Yaskawa INFORM job: A_ROOF_UPPER_0614_2_PAINT_64.JBI

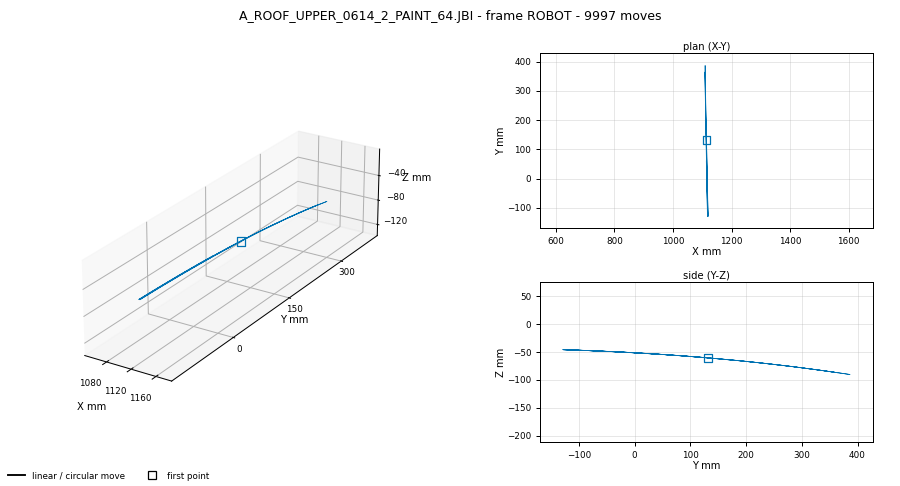
[picture p0: tool path of A_ROOF_UPPER_0614_2_PAINT_64.JBI in frame ROBOT, 9997 of 9997 moves have a stored position in this frame; points joined in program order, loops and branches not executed]
/JOB
//NAME A_ROOF_UPPER_0614_2_PAINT64
//POS
///NPOS 9997,0,0,0,0,0
///TOOL 1
///USER 0
///POSTYPE ROBOT
///RECTAN
///RCONF 1,0,0,0,0,0,0,0,0,0,0,0,0,0,0,0,0,0,0,0,0,0,0,0
C00000=1114.594,132.170,-60.301,-179.597,8.502,149.525
C00001=1114.597,131.955,-60.283,-179.599,8.499,149.525
C00002=1114.601,131.742,-60.265,-179.601,8.496,149.525
C00003=1114.606,131.528,-60.248,-179.602,8.493,149.525
C00004=1114.610,131.279,-60.226,-179.603,8.490,149.524
C00005=1114.614,131.030,-60.206,-179.605,8.487,149.524
C00006=1114.619,130.781,-60.185,-179.607,8.483,149.524
C00007=1114.624,130.532,-60.164,-179.609,8.480,149.523
C00008=1114.629,130.282,-60.143,-179.610,8.477,149.523
C00009=1114.634,130.034,-60.122,-179.613,8.473,149.523
C00010=1114.638,129.785,-60.101,-179.614,8.470,149.523
C00011=1114.643,129.535,-60.080,-179.616,8.467,149.522
C00012=1114.647,129.286,-60.059,-179.618,8.463,149.522
C00013=1114.653,129.037,-60.039,-179.619,8.460,149.522
C00014=1114.657,128.788,-60.018,-179.621,8.457,149.521
C00015=1114.662,128.539,-59.996,-179.623,8.453,149.521
C00016=1114.666,128.290,-59.976,-179.624,8.450,149.521
C00017=1114.671,128.041,-59.955,-179.626,8.447,149.521
C00018=1114.676,127.792,-59.935,-179.628,8.443,149.520
C00019=1114.681,127.543,-59.914,-179.630,8.440,149.520
C00020=1114.685,127.294,-59.893,-179.631,8.437,149.520
C00021=1114.691,127.044,-59.872,-179.634,8.433,149.519
C00022=1114.695,126.795,-59.852,-179.635,8.430,149.519
C00023=1114.700,126.547,-59.832,-179.637,8.427,149.519
C00024=1114.704,126.297,-59.810,-179.639,8.423,149.519
C00025=1114.709,126.048,-59.790,-179.640,8.420,149.518
C00026=1114.714,125.798,-59.769,-179.642,8.417,149.518
C00027=1114.718,125.549,-59.749,-179.644,8.413,149.518
C00028=1114.723,125.300,-59.728,-179.646,8.409,149.517
C00029=1114.728,125.051,-59.707,-179.647,8.407,149.517
C00030=1114.732,124.802,-59.687,-179.649,8.403,149.517
C00031=1114.737,124.553,-59.666,-179.651,8.400,149.517
C00032=1114.742,124.304,-59.646,-179.652,8.397,149.516
C00033=1114.746,124.055,-59.625,-179.655,8.393,149.516
C00034=1114.751,123.806,-59.604,-179.657,8.390,149.516
C00035=1114.756,123.557,-59.584,-179.658,8.387,149.516
C00036=1114.760,123.308,-59.564,-179.660,8.383,149.515
C00037=1114.765,123.059,-59.543,-179.662,8.380,149.515
C00038=1114.770,122.810,-59.522,-179.663,8.377,149.515
C00039=1114.774,122.561,-59.502,-179.665,8.373,149.515
C00040=1114.780,122.311,-59.482,-179.667,8.370,149.514
C00041=1114.784,122.062,-59.461,-179.669,8.366,149.514
C00042=1114.789,121.813,-59.441,-179.670,8.363,149.514
C00043=1114.794,121.564,-59.420,-179.672,8.360,149.513
C00044=1114.798,121.315,-59.399,-179.674,8.356,149.513
C00045=1114.803,121.066,-59.379,-179.675,8.353,149.513
C00046=1114.808,120.816,-59.359,-179.678,8.350,149.512
C00047=1114.813,120.567,-59.338,-179.680,8.346,149.512
C00048=1114.818,120.319,-59.318,-179.682,8.343,149.512
C00049=1114.822,120.070,-59.298,-179.683,8.340,149.512
C00050=1114.827,119.820,-59.278,-179.685,8.336,149.511
C00051=1114.832,119.571,-59.257,-179.687,8.333,149.511
C00052=1114.836,119.357,-59.240,-179.688,8.330,149.511
C00053=1114.839,119.143,-59.223,-179.690,8.327,149.511
C00054=1114.843,118.929,-59.205,-179.691,8.324,149.510
C00055=1114.848,118.715,-59.188,-179.693,8.321,149.510
C00056=1114.852,118.502,-59.171,-179.695,8.318,149.510
C00057=1114.856,118.288,-59.153,-179.696,8.315,149.510
C00058=1114.860,118.073,-59.135,-179.697,8.312,149.509
C00059=1114.864,117.860,-59.118,-179.698,8.310,149.509
C00060=1114.869,117.610,-59.098,-179.701,8.306,149.509
C00061=1114.873,117.361,-59.078,-179.703,8.303,149.509
C00062=1114.878,117.113,-59.058,-179.705,8.299,149.508
C00063=1114.883,116.863,-59.038,-179.706,8.296,149.508
C00064=1114.888,116.614,-59.017,-179.708,8.293,149.508
C00065=1114.893,116.364,-58.998,-179.710,8.289,149.508
C00066=1114.897,116.115,-58.977,-179.712,8.286,149.507
C00067=1114.902,115.867,-58.957,-179.713,8.282,149.507
C00068=1114.907,115.617,-58.937,-179.715,8.279,149.507
C00069=1114.912,115.369,-58.917,-179.717,8.275,149.506
C00070=1114.916,115.119,-58.898,-179.719,8.272,149.506
C00071=1114.921,114.870,-58.877,-179.721,8.268,149.506
C00072=1114.926,114.621,-58.858,-179.722,8.265,149.506
C00073=1114.930,114.372,-58.837,-179.724,8.262,149.505
C00074=1114.936,114.122,-58.817,-179.726,8.258,149.505
C00075=1114.941,113.874,-58.797,-179.728,8.254,149.505
C00076=1114.945,113.624,-58.777,-179.730,8.251,149.504
C00077=1114.950,113.375,-58.757,-179.731,8.248,149.504
C00078=1114.954,113.125,-58.737,-179.733,8.244,149.504
C00079=1114.959,112.876,-58.718,-179.735,8.241,149.504
C00080=1114.964,112.628,-58.698,-179.737,8.237,149.503
C00081=1114.969,112.378,-58.678,-179.739,8.233,149.503
C00082=1114.973,112.129,-58.658,-179.740,8.231,149.503
C00083=1114.978,111.880,-58.638,-179.742,8.227,149.502
C00084=1114.984,111.631,-58.619,-179.744,8.223,149.502
C00085=1114.988,111.382,-58.598,-179.746,8.220,149.502
C00086=1114.993,111.132,-58.579,-179.747,8.216,149.501
C00087=1114.997,110.883,-58.558,-179.749,8.213,149.501
C00088=1115.002,110.634,-58.539,-179.752,8.209,149.501
C00089=1115.007,110.385,-58.519,-179.754,8.206,149.501
C00090=1115.012,110.135,-58.500,-179.756,8.202,149.501
C00091=1115.016,109.886,-58.479,-179.758,8.199,149.500
C00092=1115.022,109.637,-58.460,-179.760,8.194,149.500
C00093=1115.026,109.388,-58.441,-179.762,8.190,149.500
C00094=1115.030,109.139,-58.421,-179.764,8.187,149.499
C00095=1115.036,108.890,-58.401,-179.766,8.183,149.499
C00096=1115.040,108.641,-58.382,-179.768,8.180,149.499
C00097=1115.045,108.391,-58.362,-179.770,8.176,149.499
C00098=1115.050,108.142,-58.343,-179.772,8.172,149.498
C00099=1115.055,107.893,-58.322,-179.775,8.168,149.498
C00100=1115.060,107.644,-58.303,-179.777,8.165,149.498
C00101=1115.064,107.395,-58.284,-179.778,8.161,149.497
C00102=1115.069,107.146,-58.264,-179.780,8.157,149.497
C00103=1115.074,106.896,-58.245,-179.782,8.154,149.497
C00104=1115.078,106.647,-58.225,-179.785,8.149,149.497
C00105=1115.083,106.398,-58.205,-179.787,8.146,149.496
C00106=1115.088,106.149,-58.185,-179.788,8.142,149.496
C00107=1115.093,105.900,-58.167,-179.790,8.138,149.496
C00108=1115.097,105.686,-58.150,-179.792,8.135,149.495
C00109=1115.101,105.472,-58.133,-179.793,8.132,149.495
C00110=1115.105,105.258,-58.116,-179.795,8.128,149.495
C00111=1115.110,105.043,-58.100,-179.797,8.125,149.495
C00112=1115.113,104.830,-58.083,-179.799,8.122,149.494
C00113=1115.118,104.616,-58.066,-179.800,8.119,149.494
C00114=1115.122,104.401,-58.050,-179.802,8.115,149.494
C00115=1115.126,104.188,-58.033,-179.803,8.113,149.493
C00116=1115.130,103.938,-58.014,-179.805,8.109,149.493
C00117=1115.135,103.689,-57.994,-179.807,8.105,149.493
C00118=1115.140,103.440,-57.975,-179.809,8.101,149.492
C00119=1115.144,103.191,-57.956,-179.811,8.097,149.492
C00120=1115.150,102.941,-57.937,-179.813,8.093,149.492
C00121=1115.155,102.692,-57.917,-179.814,8.089,149.491
C00122=1115.160,102.443,-57.898,-179.817,8.086,149.491
C00123=1115.164,102.194,-57.879,-179.818,8.082,149.491
C00124=1115.169,101.944,-57.859,-179.820,8.078,149.490
C00125=1115.174,101.695,-57.840,-179.822,8.074,149.490
C00126=1115.178,101.446,-57.821,-179.823,8.071,149.490
C00127=1115.183,101.197,-57.802,-179.825,8.067,149.489
C00128=1115.188,100.947,-57.782,-179.827,8.063,149.489
C00129=1115.193,100.699,-57.763,-179.829,8.059,149.488
C00130=1115.198,100.449,-57.744,-179.830,8.055,149.488
C00131=1115.202,100.200,-57.726,-179.832,8.052,149.488
C00132=1115.207,99.951,-57.706,-179.833,8.048,149.487
C00133=1115.212,99.702,-57.687,-179.836,8.044,149.487
C00134=1115.216,99.452,-57.668,-179.837,8.040,149.486
C00135=1115.222,99.203,-57.649,-179.839,8.036,149.486
C00136=1115.226,98.954,-57.630,-179.840,8.032,149.486
C00137=1115.231,98.705,-57.611,-179.842,8.029,149.485
C00138=1115.235,98.456,-57.592,-179.844,8.025,149.485
C00139=1115.241,98.206,-57.573,-179.846,8.021,149.485
C00140=1115.246,97.957,-57.554,-179.847,8.017,149.484
C00141=1115.250,97.708,-57.535,-179.849,8.013,149.484
C00142=1115.256,97.458,-57.516,-179.850,8.010,149.483
C00143=1115.260,97.209,-57.497,-179.852,8.006,149.483
C00144=1115.265,96.960,-57.478,-179.854,8.002,149.482
C00145=1115.270,96.710,-57.460,-179.855,7.998,149.482
C00146=1115.275,96.462,-57.440,-179.857,7.994,149.481
C00147=1115.279,96.212,-57.421,-179.858,7.990,149.481
C00148=1115.285,95.963,-57.403,-179.860,7.986,149.481
C00149=1115.289,95.714,-57.384,-179.862,7.982,149.480
C00150=1115.293,95.465,-57.365,-179.863,7.978,149.480
C00151=1115.298,95.215,-57.346,-179.865,7.975,149.479
C00152=1115.303,94.966,-57.327,-179.866,7.971,149.479
C00153=1115.309,94.717,-57.309,-179.868,7.967,149.478
C00154=1115.313,94.468,-57.290,-179.870,7.963,149.478
C00155=1115.318,94.218,-57.271,-179.871,7.959,149.478
C00156=1115.322,93.969,-57.252,-179.872,7.956,149.477
C00157=1115.328,93.719,-57.233,-179.874,7.952,149.477
C00158=1115.333,93.471,-57.215,-179.875,7.948,149.476
C00159=1115.337,93.221,-57.196,-179.877,7.944,149.476
C00160=1115.342,92.972,-57.177,-179.879,7.940,149.475
C00161=1115.347,92.723,-57.159,-179.880,7.936,149.475
C00162=1115.352,92.473,-57.139,-179.881,7.932,149.474
C00163=1115.357,92.224,-57.121,-179.883,7.928,149.474
C00164=1115.361,92.010,-57.105,-179.884,7.925,149.473
C00165=1115.364,91.796,-57.089,-179.885,7.922,149.473
C00166=1115.368,91.582,-57.073,-179.886,7.919,149.473
C00167=1115.373,91.368,-57.057,-179.888,7.915,149.472
C00168=1115.378,91.153,-57.041,-179.889,7.912,149.472
C00169=1115.381,90.939,-57.025,-179.890,7.909,149.472
C00170=1115.385,90.725,-57.009,-179.891,7.905,149.471
C00171=1115.390,90.512,-56.994,-179.892,7.902,149.471
C00172=1115.395,90.262,-56.975,-179.894,7.898,149.470
C00173=1115.400,90.012,-56.957,-179.896,7.894,149.470
C00174=1115.404,89.764,-56.938,-179.897,7.891,149.469
C00175=1115.409,89.514,-56.920,-179.898,7.887,149.469
C00176=1115.414,89.265,-56.901,-179.899,7.883,149.468
C00177=1115.419,89.016,-56.882,-179.901,7.879,149.468
C00178=1115.423,88.766,-56.864,-179.902,7.876,149.467
C00179=1115.429,88.517,-56.845,-179.903,7.872,149.467
C00180=1115.433,88.268,-56.827,-179.905,7.868,149.466
C00181=1115.438,88.019,-56.809,-179.906,7.864,149.466
C00182=1115.443,87.769,-56.790,-179.907,7.861,149.465
C00183=1115.448,87.520,-56.771,-179.908,7.857,149.465
C00184=1115.453,87.271,-56.753,-179.910,7.853,149.464
C00185=1115.458,87.022,-56.735,-179.911,7.848,149.464
C00186=1115.462,86.772,-56.717,-179.912,7.845,149.463
C00187=1115.467,86.523,-56.699,-179.914,7.841,149.463
C00188=1115.472,86.274,-56.680,-179.915,7.837,149.462
C00189=1115.477,86.025,-56.662,-179.916,7.833,149.462
C00190=1115.482,85.775,-56.643,-179.917,7.830,149.461
C00191=1115.486,85.526,-56.625,-179.918,7.826,149.461
C00192=1115.491,85.276,-56.607,-179.920,7.822,149.460
C00193=1115.496,85.028,-56.589,-179.920,7.819,149.460
C00194=1115.501,84.778,-56.570,-179.922,7.815,149.459
C00195=1115.506,84.529,-56.552,-179.924,7.811,149.459
C00196=1115.511,84.279,-56.534,-179.924,7.807,149.458
C00197=1115.516,84.030,-56.516,-179.926,7.803,149.458
C00198=1115.521,83.781,-56.498,-179.927,7.799,149.457
C00199=1115.525,83.531,-56.479,-179.928,7.796,149.457
C00200=1115.530,83.282,-56.461,-179.929,7.792,149.456
C00201=1115.535,83.033,-56.443,-179.930,7.789,149.456
C00202=1115.540,82.784,-56.424,-179.932,7.785,149.455
C00203=1115.545,82.535,-56.406,-179.933,7.780,149.455
C00204=1115.549,82.285,-56.388,-179.934,7.777,149.454
C00205=1115.554,82.036,-56.370,-179.935,7.773,149.453
C00206=1115.559,81.786,-56.352,-179.936,7.770,149.453
C00207=1115.564,81.537,-56.334,-179.937,7.766,149.452
C00208=1115.569,81.288,-56.316,-179.938,7.762,149.452
C00209=1115.574,81.039,-56.298,-179.939,7.758,149.451
C00210=1115.578,80.789,-56.280,-179.941,7.754,149.451
C00211=1115.583,80.540,-56.262,-179.941,7.751,149.450
C00212=1115.588,80.291,-56.244,-179.943,7.747,149.450
C00213=1115.593,80.042,-56.226,-179.943,7.743,149.449
C00214=1115.598,79.792,-56.208,-179.945,7.740,149.449
C00215=1115.603,79.543,-56.190,-179.945,7.736,149.448
C00216=1115.608,79.293,-56.172,-179.946,7.732,149.447
C00217=1115.613,79.044,-56.154,-179.947,7.729,149.447
C00218=1115.617,78.794,-56.136,-179.948,7.724,149.446
C00219=1115.622,78.545,-56.118,-179.949,7.721,149.446
C00220=1115.627,78.332,-56.102,-179.950,7.718,149.445
C00221=1115.631,78.117,-56.087,-179.951,7.715,149.445
C00222=1115.635,77.902,-56.072,-179.952,7.712,149.444
C00223=1115.640,77.688,-56.057,-179.953,7.708,149.444
C00224=1115.643,77.474,-56.040,-179.954,7.705,149.444
C00225=1115.648,77.260,-56.025,-179.955,7.702,149.443
C00226=1115.651,77.046,-56.011,-179.955,7.699,149.442
C00227=1115.656,76.832,-55.995,-179.956,7.696,149.442
C00228=1115.661,76.582,-55.977,-179.958,7.692,149.442
C00229=1115.665,76.333,-55.959,-179.959,7.688,149.441
C00230=1115.670,76.084,-55.941,-179.960,7.683,149.440
C00231=1115.675,75.834,-55.923,-179.962,7.680,149.440
C00232=1115.680,75.585,-55.905,-179.964,7.676,149.440
C00233=1115.685,75.335,-55.888,-179.965,7.672,149.439
C00234=1115.690,75.086,-55.870,-179.966,7.667,149.439
C00235=1115.695,74.837,-55.852,-179.968,7.664,149.438
C00236=1115.699,74.588,-55.835,-179.969,7.660,149.438
C00237=1115.705,74.338,-55.817,-179.970,7.656,149.437
C00238=1115.710,74.089,-55.799,-179.971,7.652,149.437
C00239=1115.714,73.840,-55.781,-179.973,7.648,149.436
C00240=1115.719,73.591,-55.764,-179.975,7.644,149.436
C00241=1115.725,73.341,-55.746,-179.976,7.640,149.435
C00242=1115.729,73.092,-55.728,-179.977,7.636,149.435
C00243=1115.734,72.843,-55.711,-179.979,7.632,149.434
C00244=1115.739,72.593,-55.694,-179.980,7.628,149.434
C00245=1115.744,72.344,-55.676,-179.982,7.624,149.433
C00246=1115.749,72.095,-55.658,-179.983,7.620,149.433
C00247=1115.754,71.845,-55.640,-179.985,7.616,149.432
C00248=1115.758,71.596,-55.623,-179.986,7.612,149.432
C00249=1115.763,71.346,-55.606,-179.987,7.608,149.431
C00250=1115.768,71.097,-55.588,-179.988,7.605,149.431
C00251=1115.773,70.848,-55.570,-179.990,7.601,149.430
C00252=1115.778,70.599,-55.553,-179.991,7.597,149.430
C00253=1115.782,70.349,-55.535,-179.993,7.593,149.429
C00254=1115.788,70.100,-55.518,-179.994,7.589,149.429
C00255=1115.793,69.850,-55.500,-179.995,7.585,149.428
C00256=1115.797,69.601,-55.483,-179.997,7.581,149.428
C00257=1115.802,69.352,-55.465,-179.998,7.577,149.427
C00258=1115.807,69.102,-55.448,-180.000,7.573,149.427
C00259=1115.812,68.853,-55.430,179.999,7.569,149.426
C00260=1115.817,68.604,-55.414,179.997,7.565,149.426
C00261=1115.822,68.355,-55.396,179.997,7.561,149.425
C00262=1115.827,68.105,-55.378,179.995,7.558,149.425
C00263=1115.832,67.856,-55.361,179.994,7.554,149.424
C00264=1115.837,67.606,-55.344,179.993,7.549,149.424
C00265=1115.842,67.357,-55.326,179.991,7.545,149.423
C00266=1115.846,67.108,-55.309,179.989,7.542,149.423
C00267=1115.851,66.858,-55.292,179.988,7.537,149.422
C00268=1115.856,66.609,-55.274,179.987,7.533,149.422
C00269=1115.861,66.359,-55.257,179.985,7.529,149.421
C00270=1115.866,66.111,-55.240,179.984,7.525,149.421
C00271=1115.871,65.861,-55.223,179.983,7.522,149.420
C00272=1115.876,65.612,-55.206,179.982,7.518,149.420
C00273=1115.881,65.362,-55.188,179.980,7.514,149.419
C00274=1115.885,65.113,-55.171,179.979,7.510,149.419
C00275=1115.891,64.863,-55.154,179.978,7.506,149.418
C00276=1115.895,64.649,-55.139,179.977,7.502,149.418
C00277=1115.899,64.435,-55.124,179.975,7.499,149.417
C00278=1115.903,64.221,-55.110,179.974,7.495,149.417
C00279=1115.908,64.006,-55.095,179.973,7.492,149.416
C00280=1115.911,63.792,-55.080,179.972,7.488,149.416
C00281=1115.916,63.578,-55.065,179.971,7.485,149.415
C00282=1115.920,63.363,-55.050,179.970,7.482,149.415
C00283=1115.924,63.149,-55.036,179.968,7.478,149.415
C00284=1115.929,62.900,-55.018,179.967,7.474,149.414
C00285=1115.934,62.650,-55.002,179.966,7.470,149.413
C00286=1115.939,62.400,-54.984,179.965,7.467,149.413
C00287=1115.944,62.152,-54.968,179.964,7.463,149.412
C00288=1115.949,61.902,-54.950,179.962,7.459,149.412
C00289=1115.953,61.653,-54.933,179.960,7.455,149.412
C00290=1115.959,61.403,-54.916,179.959,7.451,149.411
C00291=1115.964,61.154,-54.900,179.958,7.447,149.410
C00292=1115.969,60.905,-54.883,179.957,7.442,149.410
C00293=1115.973,60.655,-54.866,179.955,7.438,149.409
C00294=1115.978,60.406,-54.849,179.954,7.434,149.409
C00295=1115.983,60.156,-54.831,179.953,7.431,149.408
C00296=1115.988,59.908,-54.815,179.952,7.427,149.408
C00297=1115.993,59.658,-54.798,179.950,7.423,149.407
C00298=1115.998,59.408,-54.781,179.949,7.419,149.407
C00299=1116.003,59.159,-54.764,179.948,7.415,149.406
C00300=1116.008,58.910,-54.748,179.946,7.411,149.406
C00301=1116.012,58.660,-54.731,179.945,7.406,149.405
C00302=1116.017,58.410,-54.714,179.944,7.403,149.405
C00303=1116.023,58.162,-54.697,179.943,7.399,149.404
C00304=1116.028,57.912,-54.680,179.942,7.395,149.404
C00305=1116.032,57.662,-54.663,179.940,7.391,149.403
C00306=1116.037,57.413,-54.647,179.939,7.387,149.402
C00307=1116.043,57.164,-54.630,179.938,7.383,149.402
C00308=1116.047,56.914,-54.613,179.936,7.379,149.401
C00309=1116.052,56.665,-54.596,179.935,7.374,149.401
C00310=1116.057,56.416,-54.580,179.934,7.370,149.400
C00311=1116.062,56.166,-54.563,179.933,7.367,149.400
C00312=1116.066,55.917,-54.546,179.932,7.363,149.399
C00313=1116.072,55.668,-54.529,179.930,7.359,149.399
C00314=1116.077,55.418,-54.513,179.929,7.355,149.398
C00315=1116.081,55.169,-54.496,179.928,7.351,149.398
C00316=1116.087,54.920,-54.479,179.926,7.347,149.397
C00317=1116.091,54.670,-54.462,179.925,7.342,149.396
C00318=1116.096,54.421,-54.446,179.924,7.338,149.396
C00319=1116.102,54.171,-54.430,179.923,7.335,149.395
C00320=1116.106,53.922,-54.413,179.922,7.331,149.395
C00321=1116.112,53.673,-54.397,179.920,7.327,149.394
C00322=1116.116,53.423,-54.380,179.919,7.323,149.394
C00323=1116.121,53.173,-54.363,179.918,7.319,149.393
C00324=1116.126,52.925,-54.346,179.916,7.315,149.393
C00325=1116.131,52.675,-54.330,179.915,7.310,149.392
C00326=1116.136,52.426,-54.314,179.915,7.307,149.391
C00327=1116.141,52.176,-54.297,179.913,7.303,149.391
C00328=1116.146,51.926,-54.280,179.912,7.299,149.390
C00329=1116.151,51.677,-54.265,179.910,7.295,149.390
C00330=1116.156,51.428,-54.248,179.909,7.290,149.389
C00331=1116.161,51.179,-54.232,179.908,7.286,149.389
C00332=1116.165,50.963,-54.217,179.907,7.283,149.388
C00333=1116.169,50.750,-54.203,179.906,7.280,149.388
C00334=1116.174,50.535,-54.189,179.905,7.276,149.387
C00335=1116.178,50.321,-54.175,179.904,7.273,149.387
C00336=1116.182,50.106,-54.160,179.903,7.269,149.386
C00337=1116.186,49.892,-54.146,179.902,7.265,149.386
C00338=1116.191,49.678,-54.132,179.901,7.262,149.385
C00339=1116.195,49.463,-54.119,179.900,7.259,149.385
C00340=1116.199,49.214,-54.102,179.899,7.255,149.384
C00341=1116.205,48.965,-54.086,179.898,7.250,149.384
C00342=1116.209,48.715,-54.070,179.896,7.247,149.383
C00343=1116.215,48.466,-54.053,179.895,7.242,149.383
C00344=1116.223,48.072,-54.028,179.893,7.236,149.382
C00345=1116.230,47.678,-54.002,179.892,7.230,149.381
C00346=1116.238,47.284,-53.976,179.890,7.224,149.380
C00347=1116.245,46.890,-53.950,179.888,7.217,149.379
C00348=1116.251,46.641,-53.935,179.887,7.213,149.378
C00349=1116.255,46.391,-53.918,179.886,7.209,149.378
C00350=1116.260,46.142,-53.902,179.885,7.204,149.377
C00351=1116.266,45.893,-53.886,179.883,7.200,149.377
C00352=1116.270,45.643,-53.870,179.882,7.196,149.376
C00353=1116.276,45.394,-53.854,179.881,7.193,149.375
C00354=1116.280,45.145,-53.837,179.880,7.188,149.375
C00355=1116.286,44.895,-53.822,179.879,7.184,149.374
C00356=1116.290,44.646,-53.805,179.878,7.180,149.374
C00357=1116.295,44.396,-53.789,179.877,7.176,149.373
C00358=1116.300,44.146,-53.773,179.875,7.172,149.373
C00359=1116.305,43.897,-53.757,179.874,7.168,149.372
C00360=1116.310,43.647,-53.741,179.874,7.164,149.371
C00361=1116.315,43.399,-53.725,179.873,7.160,149.371
C00362=1116.320,43.148,-53.709,179.871,7.156,149.370
C00363=1116.325,42.900,-53.693,179.870,7.152,149.370
C00364=1116.330,42.650,-53.677,179.869,7.147,149.369
C00365=1116.335,42.400,-53.661,179.868,7.143,149.368
C00366=1116.340,42.151,-53.645,179.867,7.139,149.368
C00367=1116.345,41.901,-53.629,179.866,7.135,149.367
C00368=1116.350,41.652,-53.613,179.865,7.131,149.367
C00369=1116.356,41.403,-53.597,179.864,7.127,149.366
C00370=1116.360,41.153,-53.581,179.863,7.123,149.365
C00371=1116.366,40.904,-53.565,179.861,7.118,149.365
C00372=1116.369,40.654,-53.549,179.860,7.114,149.364
C00373=1116.375,40.405,-53.534,179.859,7.110,149.364
C00374=1116.380,40.156,-53.518,179.858,7.106,149.363
C00375=1116.385,39.906,-53.502,179.857,7.102,149.362
C00376=1116.390,39.657,-53.486,179.856,7.098,149.362
C00377=1116.395,39.407,-53.470,179.855,7.094,149.361
C00378=1116.400,39.157,-53.454,179.854,7.090,149.360
C00379=1116.405,38.909,-53.439,179.853,7.085,149.360
C00380=1116.410,38.659,-53.423,179.852,7.081,149.359
C00381=1116.415,38.409,-53.407,179.850,7.077,149.359
C00382=1116.420,38.160,-53.392,179.850,7.073,149.358
C00383=1116.426,37.910,-53.376,179.849,7.069,149.357
C00384=1116.430,37.661,-53.359,179.848,7.065,149.357
C00385=1116.435,37.412,-53.344,179.847,7.060,149.356
C00386=1116.440,37.162,-53.329,179.845,7.056,149.356
C00387=1116.445,36.912,-53.313,179.844,7.052,149.355
C00388=1116.451,36.628,-53.295,179.844,7.047,149.354
C00389=1116.456,36.344,-53.277,179.842,7.042,149.353
C00390=1116.462,36.059,-53.259,179.841,7.038,149.353
C00391=1116.468,35.775,-53.241,179.840,7.033,149.352
C00392=1116.472,35.525,-53.226,179.839,7.029,149.351
C00393=1116.478,35.275,-53.210,179.838,7.025,149.351
C00394=1116.483,35.026,-53.195,179.837,7.020,149.350
C00395=1116.488,34.777,-53.179,179.836,7.016,149.349
C00396=1116.492,34.527,-53.164,179.834,7.012,149.349
C00397=1116.498,34.277,-53.148,179.833,7.008,149.348
C00398=1116.503,34.029,-53.132,179.832,7.004,149.347
C00399=1116.508,33.778,-53.116,179.831,6.999,149.347
C00400=1116.512,33.529,-53.101,179.831,6.996,149.346
C00401=1116.518,33.280,-53.085,179.830,6.991,149.346
C00402=1116.523,33.031,-53.070,179.829,6.987,149.345
C00403=1116.528,32.781,-53.055,179.828,6.983,149.344
C00404=1116.533,32.531,-53.039,179.827,6.978,149.344
C00405=1116.538,32.282,-53.023,179.825,6.974,149.343
C00406=1116.543,32.032,-53.009,179.825,6.969,149.342
C00407=1116.548,31.783,-52.993,179.824,6.965,149.341
C00408=1116.552,31.533,-52.978,179.823,6.962,149.341
C00409=1116.558,31.284,-52.962,179.822,6.957,149.340
C00410=1116.563,31.034,-52.947,179.821,6.953,149.339
C00411=1116.568,30.785,-52.932,179.820,6.949,149.339
C00412=1116.573,30.536,-52.916,179.819,6.944,149.338
C00413=1116.578,30.286,-52.900,179.818,6.940,149.337
C00414=1116.583,30.037,-52.885,179.817,6.936,149.337
C00415=1116.588,29.787,-52.870,179.816,6.931,149.336
C00416=1116.593,29.538,-52.855,179.816,6.928,149.335
C00417=1116.598,29.288,-52.840,179.814,6.924,149.335
C00418=1116.602,29.038,-52.825,179.814,6.919,149.334
C00419=1116.608,28.789,-52.809,179.813,6.915,149.333
C00420=1116.613,28.539,-52.793,179.812,6.910,149.333
C00421=1116.618,28.290,-52.778,179.811,6.906,149.332
C00422=1116.623,28.040,-52.764,179.810,6.902,149.331
C00423=1116.628,27.791,-52.749,179.809,6.897,149.331
C00424=1116.634,27.542,-52.733,179.808,6.893,149.330
C00425=1116.638,27.292,-52.718,179.807,6.888,149.329
C00426=1116.643,27.043,-52.702,179.807,6.885,149.329
C00427=1116.648,26.793,-52.688,179.805,6.880,149.328
C00428=1116.653,26.544,-52.672,179.804,6.876,149.327
C00429=1116.658,26.294,-52.657,179.803,6.872,149.327
C00430=1116.663,26.045,-52.642,179.803,6.867,149.326
C00431=1116.668,25.795,-52.627,179.802,6.863,149.325
C00432=1116.674,25.546,-52.612,179.801,6.859,149.324
C00433=1116.678,25.297,-52.597,179.800,6.854,149.324
C00434=1116.683,25.046,-52.581,179.799,6.850,149.323
C00435=1116.688,24.797,-52.566,179.799,6.846,149.322
C00436=1116.693,24.548,-52.551,179.798,6.842,149.322
C00437=1116.698,24.298,-52.537,179.797,6.837,149.321
C00438=1116.703,24.049,-52.522,179.796,6.833,149.320
C00439=1116.708,23.799,-52.506,179.795,6.828,149.319
C00440=1116.712,23.585,-52.494,179.794,6.825,149.319
C00441=1116.717,23.370,-52.481,179.793,6.821,149.318
C00442=1116.721,23.155,-52.468,179.793,6.817,149.318
C00443=1116.726,22.942,-52.455,179.791,6.813,149.317
C00444=1116.730,22.727,-52.442,179.791,6.810,149.316
C00445=1116.734,22.512,-52.429,179.791,6.806,149.316
C00446=1116.739,22.297,-52.417,179.790,6.802,149.315
C00447=1116.743,22.082,-52.404,179.789,6.798,149.314
C00448=1116.748,21.833,-52.389,179.788,6.794,149.314
C00449=1116.753,21.583,-52.374,179.787,6.789,149.313
C00450=1116.758,21.334,-52.359,179.786,6.785,149.312
C00451=1116.763,21.085,-52.344,179.785,6.780,149.311
C00452=1116.768,20.835,-52.329,179.784,6.776,149.311
C00453=1116.773,20.586,-52.314,179.784,6.771,149.310
C00454=1116.778,20.336,-52.300,179.783,6.768,149.309
C00455=1116.783,20.087,-52.285,179.783,6.763,149.308
C00456=1116.788,19.837,-52.270,179.782,6.759,149.308
C00457=1116.794,19.587,-52.255,179.781,6.755,149.307
C00458=1116.798,19.338,-52.240,179.780,6.750,149.306
C00459=1116.803,19.088,-52.226,179.779,6.746,149.306
C00460=1116.809,18.839,-52.211,179.779,6.741,149.305
C00461=1116.814,18.589,-52.196,179.778,6.737,149.304
C00462=1116.818,18.340,-52.181,179.777,6.732,149.303
C00463=1116.823,18.090,-52.167,179.776,6.728,149.303
C00464=1116.829,17.840,-52.152,179.775,6.723,149.302
C00465=1116.833,17.591,-52.137,179.774,6.718,149.301
C00466=1116.838,17.342,-52.123,179.773,6.714,149.300
C00467=1116.843,17.093,-52.108,179.773,6.709,149.299
C00468=1116.849,16.842,-52.093,179.772,6.706,149.299
C00469=1116.854,16.593,-52.079,179.772,6.701,149.298
C00470=1116.859,16.344,-52.064,179.771,6.697,149.297
C00471=1116.864,16.095,-52.050,179.770,6.692,149.296
C00472=1116.869,15.845,-52.036,179.770,6.687,149.295
C00473=1116.874,15.596,-52.020,179.769,6.683,149.295
C00474=1116.879,15.346,-52.006,179.768,6.678,149.294
C00475=1116.884,15.096,-51.991,179.767,6.674,149.293
C00476=1116.889,14.846,-51.977,179.766,6.669,149.292
C00477=1116.894,14.597,-51.962,179.765,6.665,149.292
C00478=1116.899,14.348,-51.948,179.765,6.660,149.291
C00479=1116.904,14.098,-51.933,179.764,6.656,149.290
C00480=1116.910,13.849,-51.919,179.763,6.651,149.289
C00481=1116.915,13.600,-51.904,179.763,6.647,149.288
C00482=1116.920,13.350,-51.890,179.762,6.642,149.288
C00483=1116.925,13.100,-51.875,179.761,6.638,149.287
C00484=1116.929,12.850,-51.861,179.761,6.633,149.286
C00485=1116.934,12.601,-51.846,179.760,6.629,149.285
C00486=1116.940,12.351,-51.831,179.759,6.624,149.285
C00487=1116.945,12.102,-51.817,179.758,6.619,149.284
C00488=1116.950,11.853,-51.803,179.757,6.615,149.283
C00489=1116.955,11.603,-51.789,179.757,6.610,149.282
C00490=1116.960,11.353,-51.775,179.757,6.606,149.281
C00491=1116.965,11.103,-51.760,179.756,6.601,149.280
C00492=1116.970,10.854,-51.745,179.755,6.597,149.280
C00493=1116.975,10.605,-51.731,179.755,6.592,149.279
C00494=1116.980,10.356,-51.717,179.754,6.588,149.278
C00495=1116.985,10.106,-51.703,179.753,6.583,149.277
C00496=1116.989,9.891,-51.690,179.753,6.579,149.276
C00497=1116.994,9.676,-51.678,179.752,6.575,149.276
C00498=1116.999,9.462,-51.666,179.751,6.571,149.275
C00499=1117.002,9.247,-51.654,179.751,6.567,149.274
C00500=1117.007,9.032,-51.641,179.751,6.563,149.274
C00501=1117.012,8.818,-51.629,179.750,6.559,149.273
C00502=1117.016,8.603,-51.617,179.749,6.556,149.272
C00503=1117.020,8.388,-51.604,179.749,6.551,149.271
C00504=1117.026,8.139,-51.590,179.748,6.547,149.271
C00505=1117.030,7.890,-51.576,179.747,6.542,149.270
C00506=1117.035,7.640,-51.562,179.747,6.538,149.269
C00507=1117.040,7.390,-51.548,179.747,6.533,149.268
C00508=1117.045,7.141,-51.534,179.746,6.528,149.267
C00509=1117.050,6.891,-51.520,179.746,6.524,149.266
C00510=1117.055,6.642,-51.505,179.745,6.519,149.265
C00511=1117.060,6.392,-51.491,179.744,6.515,149.265
C00512=1117.065,6.142,-51.477,179.744,6.510,149.264
C00513=1117.071,5.893,-51.464,179.743,6.505,149.263
C00514=1117.076,5.643,-51.449,179.743,6.501,149.262
C00515=1117.081,5.393,-51.435,179.743,6.497,149.261
C00516=1117.087,5.144,-51.421,179.742,6.492,149.260
C00517=1117.092,4.895,-51.407,179.741,6.488,149.260
C00518=1117.097,4.645,-51.393,179.741,6.483,149.259
C00519=1117.102,4.395,-51.378,179.740,6.478,149.258
C00520=1117.106,4.146,-51.365,179.739,6.473,149.257
C00521=1117.111,3.897,-51.351,179.739,6.469,149.256
C00522=1117.117,3.646,-51.337,179.739,6.465,149.255
C00523=1117.122,3.397,-51.323,179.738,6.460,149.255
C00524=1117.127,3.148,-51.309,179.737,6.456,149.254
C00525=1117.132,2.898,-51.295,179.737,6.451,149.253
C00526=1117.137,2.648,-51.281,179.736,6.446,149.252
C00527=1117.142,2.400,-51.267,179.735,6.442,149.251
C00528=1117.147,2.149,-51.254,179.735,6.437,149.250
C00529=1117.152,1.900,-51.239,179.734,6.433,149.249
C00530=1117.158,1.651,-51.225,179.734,6.429,149.249
C00531=1117.162,1.401,-51.211,179.733,6.424,149.248
C00532=1117.167,1.151,-51.198,179.733,6.420,149.247
C00533=1117.173,0.902,-51.184,179.732,6.415,149.246
C00534=1117.178,0.652,-51.170,179.732,6.410,149.245
C00535=1117.182,0.402,-51.156,179.731,6.406,149.245
C00536=1117.188,0.153,-51.143,179.730,6.401,149.244
C00537=1117.193,-0.097,-51.129,179.730,6.396,149.243
C00538=1117.198,-0.346,-51.115,179.730,6.392,149.242
C00539=1117.203,-0.596,-51.101,179.729,6.388,149.241
C00540=1117.208,-0.846,-51.087,179.728,6.383,149.240
C00541=1117.213,-1.094,-51.074,179.728,6.379,149.239
C00542=1117.218,-1.345,-51.060,179.727,6.374,149.239
C00543=1117.223,-1.594,-51.046,179.726,6.370,149.238
C00544=1117.229,-1.843,-51.032,179.726,6.365,149.237
C00545=1117.233,-2.093,-51.019,179.725,6.360,149.236
C00546=1117.239,-2.342,-51.005,179.725,6.357,149.235
C00547=1117.244,-2.592,-50.991,179.724,6.352,149.235
C00548=1117.248,-2.842,-50.978,179.724,6.347,149.234
C00549=1117.254,-3.091,-50.964,179.723,6.343,149.233
C00550=1117.259,-3.342,-50.950,179.722,6.338,149.232
C00551=1117.265,-3.591,-50.937,179.722,6.333,149.231
C00552=1117.269,-3.806,-50.925,179.721,6.330,149.231
C00553=1117.273,-4.020,-50.913,179.720,6.326,149.230
C00554=1117.278,-4.235,-50.901,179.720,6.322,149.229
C00555=1117.282,-4.450,-50.890,179.720,6.318,149.228
C00556=1117.287,-4.665,-50.878,179.719,6.314,149.228
C00557=1117.291,-4.879,-50.866,179.719,6.310,149.227
C00558=1117.295,-5.094,-50.854,179.718,6.307,149.226
C00559=1117.300,-5.309,-50.843,179.717,6.302,149.226
C00560=1117.305,-5.559,-50.830,179.717,6.298,149.225
C00561=1117.310,-5.808,-50.816,179.716,6.293,149.224
C00562=1117.315,-6.058,-50.803,179.716,6.289,149.223
C00563=1117.320,-6.307,-50.789,179.715,6.285,149.222
C00564=1117.325,-6.557,-50.776,179.715,6.280,149.221
C00565=1117.330,-6.806,-50.762,179.714,6.276,149.221
C00566=1117.336,-7.056,-50.749,179.713,6.271,149.220
C00567=1117.340,-7.305,-50.735,179.713,6.266,149.219
C00568=1117.346,-7.555,-50.722,179.712,6.261,149.218
C00569=1117.351,-7.805,-50.708,179.711,6.257,149.218
C00570=1117.356,-8.054,-50.695,179.711,6.252,149.217
C00571=1117.361,-8.304,-50.682,179.710,6.248,149.216
C00572=1117.366,-8.553,-50.668,179.709,6.243,149.215
C00573=1117.372,-8.803,-50.655,179.709,6.239,149.214
C00574=1117.376,-9.052,-50.641,179.709,6.235,149.213
C00575=1117.382,-9.302,-50.628,179.708,6.230,149.213
C00576=1117.386,-9.552,-50.615,179.707,6.226,149.212
C00577=1117.392,-9.801,-50.601,179.707,6.221,149.211
C00578=1117.396,-10.051,-50.588,179.706,6.216,149.210
C00579=1117.402,-10.300,-50.575,179.705,6.212,149.209
C00580=1117.406,-10.550,-50.561,179.705,6.207,149.208
C00581=1117.412,-10.799,-50.548,179.704,6.202,149.207
C00582=1117.417,-11.049,-50.535,179.703,6.198,149.207
C00583=1117.423,-11.299,-50.522,179.703,6.193,149.206
C00584=1117.427,-11.549,-50.508,179.702,6.189,149.205
C00585=1117.433,-11.798,-50.495,179.702,6.184,149.204
C00586=1117.438,-12.047,-50.483,179.701,6.179,149.203
C00587=1117.443,-12.298,-50.469,179.700,6.175,149.203
C00588=1117.448,-12.546,-50.456,179.700,6.170,149.202
C00589=1117.452,-12.796,-50.443,179.699,6.166,149.201
C00590=1117.458,-13.046,-50.430,179.698,6.161,149.200
C00591=1117.463,-13.295,-50.417,179.698,6.156,149.199
C00592=1117.468,-13.545,-50.403,179.697,6.151,149.198
C00593=1117.473,-13.794,-50.390,179.696,6.147,149.198
C00594=1117.478,-14.044,-50.377,179.696,6.142,149.197
C00595=1117.484,-14.294,-50.364,179.695,6.138,149.196
C00596=1117.489,-14.543,-50.351,179.695,6.133,149.195
C00597=1117.494,-14.794,-50.338,179.694,6.129,149.194
C00598=1117.499,-15.042,-50.324,179.693,6.124,149.193
C00599=1117.504,-15.292,-50.312,179.693,6.119,149.193
C00600=1117.509,-15.542,-50.298,179.692,6.114,149.192
C00601=1117.515,-15.791,-50.286,179.691,6.110,149.191
C00602=1117.519,-16.041,-50.273,179.691,6.105,149.190
C00603=1117.525,-16.291,-50.260,179.690,6.101,149.189
C00604=1117.530,-16.540,-50.247,179.690,6.096,149.188
C00605=1117.535,-16.790,-50.234,179.689,6.092,149.188
C00606=1117.540,-17.040,-50.221,179.689,6.087,149.187
C00607=1117.546,-17.289,-50.208,179.688,6.082,149.186
C00608=1117.550,-17.505,-50.197,179.688,6.079,149.185
C00609=1117.554,-17.719,-50.186,179.687,6.074,149.184
C00610=1117.559,-17.933,-50.174,179.687,6.070,149.184
C00611=1117.563,-18.149,-50.163,179.686,6.066,149.183
C00612=1117.568,-18.364,-50.152,179.685,6.062,149.182
C00613=1117.572,-18.578,-50.141,179.686,6.058,149.181
C00614=1117.576,-18.793,-50.130,179.685,6.054,149.181
C00615=1117.581,-19.008,-50.118,179.684,6.051,149.180
C00616=1117.586,-19.258,-50.107,179.684,6.046,149.179
C00617=1117.591,-19.508,-50.094,179.683,6.040,149.178
C00618=1117.596,-19.757,-50.081,179.682,6.036,149.177
C00619=1117.602,-20.007,-50.068,179.682,6.031,149.176
C00620=1117.607,-20.256,-50.055,179.681,6.026,149.176
C00621=1117.611,-20.506,-50.042,179.680,6.022,149.175
C00622=1117.616,-20.755,-50.030,179.680,6.017,149.174
C00623=1117.622,-21.005,-50.016,179.679,6.012,149.173
C00624=1117.627,-21.254,-50.004,179.679,6.008,149.172
C00625=1117.632,-21.504,-49.991,179.678,6.003,149.171
C00626=1117.637,-21.754,-49.978,179.678,5.998,149.170
C00627=1117.642,-22.003,-49.966,179.677,5.993,149.170
C00628=1117.648,-22.253,-49.953,179.677,5.989,149.169
C00629=1117.653,-22.503,-49.940,179.675,5.983,149.168
C00630=1117.658,-22.753,-49.928,179.675,5.979,149.167
C00631=1117.663,-23.002,-49.915,179.674,5.974,149.166
C00632=1117.668,-23.251,-49.902,179.674,5.969,149.165
C00633=1117.673,-23.501,-49.890,179.673,5.965,149.164
C00634=1117.679,-23.752,-49.877,179.673,5.960,149.163
C00635=1117.684,-24.001,-49.864,179.672,5.955,149.163
C00636=1117.689,-24.250,-49.852,179.672,5.950,149.162
C00637=1117.694,-24.500,-49.839,179.671,5.945,149.161
C00638=1117.700,-24.749,-49.827,179.670,5.940,149.160
C00639=1117.704,-24.999,-49.814,179.670,5.935,149.159
C00640=1117.709,-25.249,-49.802,179.669,5.931,149.158
C00641=1117.715,-25.498,-49.789,179.669,5.926,149.157
C00642=1117.720,-25.748,-49.777,179.668,5.921,149.156
C00643=1117.725,-25.997,-49.765,179.668,5.916,149.155
C00644=1117.731,-26.247,-49.751,179.669,5.912,149.154
C00645=1117.736,-26.498,-49.739,179.669,5.908,149.153
C00646=1117.741,-26.747,-49.727,179.670,5.903,149.152
C00647=1117.746,-26.996,-49.714,179.670,5.899,149.151
C00648=1117.751,-27.246,-49.701,179.671,5.895,149.150
C00649=1117.757,-27.496,-49.690,179.671,5.891,149.149
C00650=1117.762,-27.745,-49.677,179.671,5.887,149.148
C00651=1117.767,-27.994,-49.664,179.672,5.883,149.147
C00652=1117.772,-28.245,-49.652,179.672,5.879,149.146
C00653=1117.777,-28.494,-49.639,179.673,5.874,149.145
C00654=1117.782,-28.743,-49.627,179.673,5.870,149.144
C00655=1117.787,-28.993,-49.615,179.674,5.866,149.143
C00656=1117.792,-29.243,-49.602,179.673,5.861,149.142
C00657=1117.798,-29.493,-49.591,179.673,5.857,149.141
C00658=1117.803,-29.742,-49.578,179.673,5.853,149.140
C00659=1117.808,-29.992,-49.565,179.674,5.849,149.139
C00660=1117.813,-30.242,-49.553,179.674,5.844,149.138
C00661=1117.818,-30.491,-49.540,179.674,5.840,149.137
C00662=1117.824,-30.741,-49.529,179.674,5.836,149.136
C00663=1117.829,-30.990,-49.516,179.673,5.832,149.135
C00664=1117.833,-31.205,-49.506,179.673,5.828,149.134
C00665=1117.838,-31.420,-49.495,179.673,5.824,149.134
C00666=1117.842,-31.635,-49.484,179.673,5.820,149.133
C00667=1117.847,-31.851,-49.474,179.673,5.817,149.132
C00668=1117.851,-32.065,-49.463,179.673,5.813,149.131
C00669=1117.856,-32.280,-49.452,179.673,5.809,149.131
C00670=1117.860,-32.495,-49.442,179.673,5.805,149.130
C00671=1117.864,-32.709,-49.432,179.673,5.802,149.129
C00672=1117.869,-32.960,-49.419,179.672,5.797,149.128
C00673=1117.874,-33.209,-49.407,179.672,5.793,149.127
C00674=1117.879,-33.459,-49.395,179.672,5.788,149.126
C00675=1117.885,-33.708,-49.382,179.671,5.784,149.126
C00676=1117.890,-33.958,-49.370,179.670,5.779,149.125
C00677=1117.895,-34.208,-49.358,179.671,5.775,149.124
C00678=1117.901,-34.458,-49.346,179.670,5.771,149.123
C00679=1117.906,-34.707,-49.333,179.670,5.766,149.122
C00680=1117.911,-34.957,-49.321,179.669,5.761,149.121
C00681=1117.916,-35.206,-49.309,179.668,5.757,149.120
C00682=1117.921,-35.456,-49.298,179.668,5.752,149.119
C00683=1117.926,-35.706,-49.286,179.667,5.747,149.119
C00684=1117.931,-35.955,-49.273,179.666,5.743,149.118
C00685=1117.937,-36.205,-49.261,179.666,5.738,149.117
C00686=1117.942,-36.454,-49.249,179.665,5.733,149.116
C00687=1117.947,-36.704,-49.237,179.665,5.729,149.115
C00688=1117.952,-36.954,-49.225,179.664,5.724,149.114
C00689=1117.957,-37.203,-49.213,179.663,5.719,149.114
C00690=1117.963,-37.453,-49.201,179.662,5.714,149.113
C00691=1117.968,-37.703,-49.189,179.662,5.710,149.112
C00692=1117.973,-37.952,-49.176,179.661,5.704,149.111
C00693=1117.979,-38.202,-49.165,179.660,5.700,149.110
C00694=1117.983,-38.452,-49.153,179.659,5.695,149.110
C00695=1117.989,-38.701,-49.141,179.658,5.690,149.109
C00696=1117.994,-38.951,-49.129,179.657,5.685,149.108
C00697=1117.999,-39.201,-49.117,179.656,5.680,149.107
C00698=1118.004,-39.451,-49.106,179.655,5.675,149.106
C00699=1118.009,-39.700,-49.093,179.654,5.670,149.105
C00700=1118.015,-39.950,-49.081,179.653,5.665,149.105
C00701=1118.020,-40.200,-49.069,179.652,5.660,149.104
C00702=1118.025,-40.450,-49.058,179.651,5.654,149.103
C00703=1118.030,-40.698,-49.046,179.650,5.649,149.102
C00704=1118.036,-40.948,-49.034,179.649,5.644,149.101
C00705=1118.041,-41.198,-49.022,179.648,5.639,149.101
C00706=1118.046,-41.448,-49.011,179.647,5.634,149.100
C00707=1118.051,-41.698,-48.999,179.646,5.628,149.099
C00708=1118.057,-41.948,-48.987,179.644,5.623,149.098
C00709=1118.061,-42.197,-48.975,179.643,5.617,149.097
C00710=1118.067,-42.446,-48.963,179.642,5.612,149.096
C00711=1118.072,-42.696,-48.951,179.641,5.607,149.096
C00712=1118.077,-42.945,-48.940,179.639,5.600,149.095
C00713=1118.083,-43.195,-48.928,179.639,5.596,149.094
C00714=1118.088,-43.445,-48.917,179.639,5.591,149.093
C00715=1118.093,-43.695,-48.905,179.639,5.586,149.092
C00716=1118.098,-43.945,-48.893,179.640,5.582,149.091
C00717=1118.103,-44.194,-48.882,179.639,5.577,149.090
C00718=1118.109,-44.444,-48.870,179.640,5.573,149.088
C00719=1118.114,-44.693,-48.859,179.640,5.568,149.087
C00720=1118.119,-44.908,-48.849,179.640,5.564,149.086
C00721=1118.123,-45.123,-48.839,179.640,5.560,149.086
C00722=1118.128,-45.338,-48.829,179.641,5.556,149.085
C00723=1118.132,-45.553,-48.818,179.641,5.552,149.084
C00724=1118.137,-45.769,-48.809,179.640,5.547,149.083
C00725=1118.141,-45.983,-48.799,179.641,5.543,149.082
C00726=1118.145,-46.198,-48.789,179.641,5.539,149.081
C00727=1118.150,-46.413,-48.779,179.641,5.535,149.080
C00728=1118.155,-46.663,-48.767,179.642,5.531,149.079
C00729=1118.160,-46.913,-48.755,179.642,5.526,149.078
C00730=1118.165,-47.163,-48.744,179.642,5.521,149.077
C00731=1118.171,-47.413,-48.732,179.642,5.517,149.076
C00732=1118.176,-47.661,-48.721,179.642,5.511,149.075
C00733=1118.181,-47.911,-48.709,179.643,5.507,149.073
C00734=1118.186,-48.161,-48.698,179.642,5.502,149.072
C00735=1118.192,-48.412,-48.687,179.642,5.497,149.071
C00736=1118.196,-48.661,-48.676,179.643,5.493,149.070
C00737=1118.202,-48.910,-48.664,179.643,5.488,149.069
C00738=1118.207,-49.160,-48.653,179.643,5.484,149.068
C00739=1118.213,-49.410,-48.641,179.643,5.479,149.067
C00740=1118.217,-49.660,-48.630,179.643,5.474,149.066
C00741=1118.223,-49.909,-48.618,179.644,5.470,149.065
C00742=1118.228,-50.158,-48.607,179.644,5.464,149.064
C00743=1118.233,-50.408,-48.595,179.644,5.460,149.063
C00744=1118.238,-50.659,-48.584,179.644,5.455,149.061
C00745=1118.244,-50.908,-48.573,179.644,5.450,149.061
C00746=1118.249,-51.158,-48.562,179.645,5.446,149.059
C00747=1118.255,-51.407,-48.550,179.645,5.441,149.058
C00748=1118.259,-51.657,-48.538,179.645,5.437,149.057
C00749=1118.265,-51.906,-48.528,179.645,5.432,149.056
C00750=1118.270,-52.157,-48.516,179.645,5.427,149.055
C00751=1118.275,-52.406,-48.505,179.645,5.423,149.054
C00752=1118.280,-52.656,-48.493,179.645,5.417,149.053
C00753=1118.286,-52.905,-48.482,179.646,5.413,149.052
C00754=1118.291,-53.155,-48.470,179.646,5.408,149.051
C00755=1118.296,-53.405,-48.460,179.646,5.403,149.050
C00756=1118.301,-53.654,-48.449,179.646,5.399,149.049
C00757=1118.307,-53.904,-48.437,179.646,5.394,149.048
C00758=1118.311,-54.154,-48.426,179.647,5.390,149.047
C00759=1118.318,-54.404,-48.415,179.647,5.385,149.045
C00760=1118.323,-54.653,-48.404,179.646,5.380,149.044
C00761=1118.327,-54.903,-48.392,179.647,5.376,149.043
C00762=1118.333,-55.153,-48.380,179.647,5.370,149.042
C00763=1118.338,-55.402,-48.370,179.647,5.367,149.041
C00764=1118.343,-55.652,-48.359,179.647,5.361,149.040
C00765=1118.348,-55.902,-48.347,179.647,5.356,149.039
C00766=1118.354,-56.151,-48.337,179.648,5.352,149.038
C00767=1118.359,-56.401,-48.326,179.648,5.347,149.037
C00768=1118.364,-56.651,-48.314,179.648,5.343,149.036
C00769=1118.370,-56.901,-48.303,179.648,5.338,149.035
C00770=1118.374,-57.150,-48.292,179.649,5.334,149.034
C00771=1118.380,-57.400,-48.280,179.648,5.329,149.033
C00772=1118.385,-57.650,-48.270,179.648,5.324,149.032
C00773=1118.390,-57.899,-48.259,179.649,5.319,149.030
C00774=1118.396,-58.149,-48.247,179.649,5.315,149.030
C00775=1118.401,-58.399,-48.237,179.649,5.310,149.028
C00776=1118.405,-58.614,-48.227,179.649,5.306,149.027
C00777=1118.410,-58.829,-48.217,179.649,5.302,149.027
C00778=1118.414,-59.044,-48.207,179.649,5.298,149.026
C00779=1118.418,-59.259,-48.199,179.650,5.294,149.025
C00780=1118.423,-59.474,-48.189,179.650,5.290,149.024
C00781=1118.427,-59.690,-48.179,179.650,5.286,149.023
C00782=1118.433,-59.904,-48.170,179.650,5.282,149.022
C00783=1118.437,-60.119,-48.160,179.650,5.278,149.021
C00784=1118.442,-60.369,-48.150,179.649,5.272,149.020
C00785=1118.447,-60.619,-48.139,179.649,5.268,149.019
C00786=1118.453,-60.869,-48.128,179.648,5.262,149.018
C00787=1118.458,-61.119,-48.117,179.648,5.257,149.017
C00788=1118.463,-61.367,-48.106,179.647,5.252,149.016
C00789=1118.468,-61.618,-48.095,179.646,5.247,149.015
C00790=1118.474,-61.867,-48.083,179.645,5.241,149.015
C00791=1118.479,-62.117,-48.073,179.645,5.237,149.014
C00792=1118.484,-62.367,-48.062,179.644,5.231,149.013
C00793=1118.489,-62.616,-48.051,179.644,5.226,149.012
C00794=1118.494,-62.867,-48.041,179.644,5.221,149.011
C00795=1118.500,-63.115,-48.030,179.643,5.216,149.010
C00796=1118.505,-63.366,-48.019,179.642,5.211,149.009
C00797=1118.511,-63.615,-48.008,179.641,5.205,149.008
C00798=1118.516,-63.865,-47.997,179.641,5.200,149.007
C00799=1118.520,-64.115,-47.986,179.640,5.195,149.006
C00800=1118.526,-64.364,-47.976,179.640,5.190,149.005
C00801=1118.531,-64.615,-47.965,179.639,5.184,149.004
C00802=1118.536,-64.864,-47.954,179.639,5.179,149.003
C00803=1118.542,-65.114,-47.943,179.639,5.174,149.002
C00804=1118.547,-65.364,-47.933,179.638,5.169,149.001
C00805=1118.552,-65.613,-47.922,179.638,5.164,149.000
C00806=1118.558,-65.863,-47.911,179.637,5.158,148.999
C00807=1118.563,-66.113,-47.901,179.637,5.153,148.998
C00808=1118.568,-66.362,-47.890,179.637,5.148,148.997
C00809=1118.573,-66.612,-47.879,179.636,5.143,148.996
C00810=1118.579,-66.862,-47.869,179.636,5.138,148.995
C00811=1118.583,-67.111,-47.858,179.636,5.133,148.994
C00812=1118.589,-67.361,-47.848,179.635,5.127,148.993
C00813=1118.595,-67.610,-47.837,179.635,5.122,148.992
C00814=1118.600,-67.861,-47.827,179.635,5.117,148.991
C00815=1118.605,-68.110,-47.816,179.634,5.111,148.990
C00816=1118.610,-68.360,-47.805,179.634,5.106,148.989
C00817=1118.615,-68.609,-47.795,179.633,5.101,148.988
C00818=1118.620,-68.860,-47.785,179.633,5.095,148.986
C00819=1118.626,-69.109,-47.774,179.633,5.091,148.986
C00820=1118.631,-69.359,-47.763,179.633,5.086,148.984
C00821=1118.636,-69.608,-47.753,179.632,5.080,148.983
C00822=1118.642,-69.858,-47.743,179.632,5.075,148.982
C00823=1118.647,-70.108,-47.732,179.632,5.070,148.981
C00824=1118.653,-70.358,-47.722,179.631,5.064,148.980
C00825=1118.658,-70.608,-47.711,179.631,5.059,148.979
C00826=1118.663,-70.857,-47.700,179.631,5.054,148.978
C00827=1118.668,-71.106,-47.690,179.631,5.049,148.977
C00828=1118.673,-71.357,-47.680,179.631,5.043,148.976
C00829=1118.679,-71.606,-47.669,179.631,5.038,148.975
C00830=1118.684,-71.856,-47.659,179.630,5.033,148.974
C00831=1118.690,-72.106,-47.649,179.631,5.028,148.973
C00832=1118.694,-72.322,-47.639,179.630,5.023,148.972
C00833=1118.699,-72.536,-47.631,179.630,5.019,148.971
C00834=1118.703,-72.751,-47.622,179.630,5.015,148.970
C00835=1118.707,-72.967,-47.613,179.630,5.010,148.969
C00836=1118.713,-73.181,-47.604,179.629,5.005,148.968
C00837=1118.717,-73.397,-47.595,179.630,5.001,148.967
C00838=1118.721,-73.612,-47.586,179.630,4.996,148.966
C00839=1118.726,-73.827,-47.577,179.630,4.992,148.965
C00840=1118.731,-74.077,-47.567,179.630,4.986,148.964
C00841=1118.736,-74.326,-47.557,179.629,4.981,148.963
C00842=1118.742,-74.576,-47.547,179.629,4.976,148.962
C00843=1118.747,-74.826,-47.536,179.629,4.971,148.960
C00844=1118.752,-75.076,-47.526,179.630,4.966,148.959
C00845=1118.758,-75.326,-47.516,179.630,4.961,148.958
C00846=1118.763,-75.576,-47.506,179.629,4.955,148.957
C00847=1118.769,-75.826,-47.496,179.629,4.950,148.956
C00848=1118.774,-76.075,-47.486,179.629,4.945,148.955
C00849=1118.779,-76.324,-47.476,179.629,4.940,148.954
C00850=1118.784,-76.575,-47.465,179.629,4.934,148.952
C00851=1118.790,-76.824,-47.455,179.630,4.929,148.951
C00852=1118.796,-77.074,-47.445,179.630,4.924,148.950
C00853=1118.800,-77.324,-47.435,179.630,4.919,148.949
C00854=1118.805,-77.573,-47.425,179.630,4.914,148.948
C00855=1118.811,-77.823,-47.414,179.630,4.909,148.947
C00856=1118.817,-78.072,-47.404,179.630,4.903,148.945
C00857=1118.822,-78.323,-47.394,179.630,4.898,148.944
C00858=1118.827,-78.572,-47.385,179.630,4.892,148.943
C00859=1118.832,-78.822,-47.375,179.630,4.887,148.942
C00860=1118.838,-79.071,-47.364,179.630,4.882,148.941
C00861=1118.843,-79.322,-47.354,179.631,4.877,148.940
C00862=1118.848,-79.571,-47.344,179.631,4.872,148.938
C00863=1118.854,-79.821,-47.335,179.631,4.867,148.937
C00864=1118.859,-80.071,-47.324,179.631,4.861,148.936
C00865=1118.864,-80.321,-47.314,179.631,4.856,148.935
C00866=1118.869,-80.570,-47.304,179.631,4.851,148.934
C00867=1118.875,-80.820,-47.294,179.631,4.846,148.933
C00868=1118.881,-81.070,-47.285,179.632,4.841,148.931
C00869=1118.886,-81.319,-47.275,179.632,4.837,148.930
C00870=1118.891,-81.569,-47.264,179.633,4.831,148.929
C00871=1118.896,-81.819,-47.254,179.633,4.826,148.928
C00872=1118.901,-82.069,-47.245,179.633,4.821,148.927
C00873=1118.907,-82.318,-47.235,179.633,4.816,148.926
C00874=1118.912,-82.569,-47.224,179.633,4.811,148.924
C00875=1118.917,-82.818,-47.216,179.633,4.806,148.923
C00876=1118.923,-83.068,-47.205,179.634,4.800,148.922
C00877=1118.928,-83.317,-47.195,179.634,4.795,148.921
C00878=1118.933,-83.567,-47.186,179.634,4.790,148.919
C00879=1118.939,-83.817,-47.176,179.635,4.785,148.918
C00880=1118.944,-84.067,-47.166,179.635,4.780,148.917
C00881=1118.949,-84.316,-47.156,179.636,4.775,148.916
C00882=1118.955,-84.567,-47.146,179.636,4.770,148.915
C00883=1118.960,-84.816,-47.137,179.636,4.765,148.914
C00884=1118.965,-85.065,-47.127,179.637,4.760,148.912
C00885=1118.971,-85.315,-47.117,179.637,4.755,148.911
C00886=1118.975,-85.565,-47.107,179.638,4.750,148.910
C00887=1118.981,-85.816,-47.098,179.638,4.745,148.909
C00888=1118.986,-86.030,-47.089,179.638,4.741,148.908
C00889=1118.990,-86.245,-47.081,179.639,4.736,148.907
C00890=1118.995,-86.461,-47.072,179.639,4.732,148.906
C00891=1118.999,-86.676,-47.064,179.639,4.727,148.904
C00892=1119.004,-86.891,-47.056,179.639,4.723,148.903
C00893=1119.009,-87.106,-47.047,179.640,4.719,148.902
C00894=1119.013,-87.322,-47.039,179.640,4.715,148.901
C00895=1119.017,-87.537,-47.030,179.641,4.710,148.900
C00896=1119.023,-87.787,-47.021,179.641,4.705,148.899
C00897=1119.028,-88.036,-47.011,179.642,4.700,148.898
C00898=1119.034,-88.286,-47.002,179.642,4.696,148.897
C00899=1119.039,-88.536,-46.991,179.643,4.691,148.895
C00900=1119.044,-88.786,-46.982,179.643,4.686,148.894
C00901=1119.050,-89.036,-46.972,179.644,4.681,148.893
C00902=1119.055,-89.286,-46.963,179.644,4.676,148.892
C00903=1119.061,-89.535,-46.953,179.644,4.670,148.890
C00904=1119.066,-89.785,-46.944,179.645,4.666,148.889
C00905=1119.071,-90.035,-46.934,179.645,4.661,148.888
C00906=1119.077,-90.284,-46.925,179.647,4.656,148.887
C00907=1119.082,-90.534,-46.915,179.647,4.651,148.885
C00908=1119.087,-90.784,-46.906,179.648,4.647,148.884
C00909=1119.092,-91.034,-46.895,179.648,4.642,148.883
C00910=1119.097,-91.284,-46.886,179.648,4.636,148.882
C00911=1119.102,-91.533,-46.877,179.649,4.632,148.881
C00912=1119.108,-91.783,-46.867,179.650,4.626,148.879
C00913=1119.113,-92.033,-46.858,179.650,4.622,148.878
C00914=1119.119,-92.283,-46.848,179.651,4.617,148.877
C00915=1119.124,-92.532,-46.839,179.651,4.613,148.876
C00916=1119.130,-92.782,-46.829,179.652,4.608,148.875
C00917=1119.135,-93.032,-46.820,179.653,4.603,148.873
C00918=1119.140,-93.282,-46.810,179.654,4.598,148.872
C00919=1119.146,-93.531,-46.801,179.654,4.593,148.871
C00920=1119.151,-93.781,-46.792,179.655,4.589,148.870
C00921=1119.156,-94.031,-46.782,179.655,4.584,148.868
C00922=1119.162,-94.281,-46.773,179.656,4.579,148.867
C00923=1119.167,-94.530,-46.763,179.656,4.574,148.866
C00924=1119.172,-94.780,-46.754,179.657,4.569,148.865
C00925=1119.178,-95.030,-46.744,179.657,4.564,148.863
C00926=1119.183,-95.279,-46.735,179.657,4.560,148.862
C00927=1119.188,-95.529,-46.726,179.657,4.554,148.861
C00928=1119.194,-95.779,-46.716,179.658,4.550,148.860
C00929=1119.199,-96.029,-46.707,179.658,4.545,148.859
C00930=1119.205,-96.279,-46.697,179.658,4.540,148.858
C00931=1119.210,-96.528,-46.688,179.659,4.535,148.857
C00932=1119.215,-96.778,-46.679,179.659,4.530,148.855
C00933=1119.221,-97.028,-46.669,179.660,4.525,148.854
C00934=1119.226,-97.278,-46.661,179.660,4.520,148.853
C00935=1119.231,-97.527,-46.651,179.660,4.515,148.852
C00936=1119.237,-97.777,-46.641,179.661,4.510,148.851
C00937=1119.242,-98.027,-46.633,179.661,4.505,148.849
C00938=1119.247,-98.276,-46.623,179.661,4.500,148.848
C00939=1119.253,-98.527,-46.613,179.662,4.495,148.847
C00940=1119.258,-98.776,-46.605,179.662,4.490,148.846
C00941=1119.263,-99.026,-46.596,179.663,4.485,148.845
C00942=1119.269,-99.276,-46.585,179.662,4.481,148.844
C00943=1119.274,-99.526,-46.577,179.662,4.475,148.843
C00944=1119.279,-99.741,-46.569,179.663,4.471,148.841
C00945=1119.283,-99.957,-46.561,179.664,4.467,148.840
C00946=1119.288,-100.172,-46.553,179.663,4.462,148.839
C00947=1119.293,-100.388,-46.545,179.664,4.458,148.838
C00948=1119.297,-100.602,-46.536,179.664,4.454,148.837
C00949=1119.301,-100.818,-46.528,179.664,4.449,148.836
C00950=1119.306,-101.033,-46.521,179.664,4.445,148.835
C00951=1119.311,-101.248,-46.513,179.665,4.441,148.834
C00952=1119.316,-101.498,-46.504,179.665,4.436,148.833
C00953=1119.322,-101.748,-46.495,179.665,4.431,148.832
C00954=1119.327,-101.998,-46.486,179.665,4.426,148.831
C00955=1119.332,-102.248,-46.477,179.666,4.421,148.830
C00956=1119.337,-102.497,-46.467,179.666,4.416,148.828
C00957=1119.342,-102.747,-46.459,179.667,4.411,148.827
C00958=1119.348,-102.997,-46.449,179.667,4.406,148.826
C00959=1119.353,-103.247,-46.440,179.667,4.401,148.825
C00960=1119.359,-103.497,-46.431,179.667,4.396,148.824
C00961=1119.364,-103.746,-46.423,179.668,4.390,148.822
C00962=1119.370,-103.996,-46.413,179.668,4.386,148.821
C00963=1119.376,-104.246,-46.404,179.669,4.381,148.820
C00964=1119.380,-104.495,-46.395,179.669,4.376,148.819
C00965=1119.386,-104.745,-46.386,179.669,4.371,148.818
C00966=1119.391,-104.995,-46.377,179.669,4.365,148.817
C00967=1119.396,-105.245,-46.368,179.670,4.360,148.815
C00968=1119.402,-105.495,-46.359,179.670,4.355,148.814
C00969=1119.407,-105.745,-46.350,179.669,4.350,148.813
C00970=1119.413,-105.994,-46.341,179.670,4.346,148.812
C00971=1119.418,-106.244,-46.332,179.671,4.341,148.811
C00972=1119.423,-106.494,-46.323,179.671,4.336,148.810
C00973=1119.428,-106.744,-46.314,179.671,4.330,148.808
C00974=1119.434,-106.994,-46.305,179.671,4.325,148.807
C00975=1119.439,-107.244,-46.296,179.672,4.320,148.806
C00976=1119.445,-107.493,-46.287,179.672,4.315,148.805
C00977=1119.450,-107.743,-46.279,179.672,4.310,148.804
C00978=1119.455,-107.992,-46.270,179.672,4.305,148.802
C00979=1119.461,-108.242,-46.261,179.672,4.299,148.801
C00980=1119.466,-108.492,-46.252,179.673,4.294,148.800
C00981=1119.471,-108.742,-46.243,179.673,4.289,148.799
C00982=1119.477,-108.991,-46.234,179.673,4.284,148.798
C00983=1119.482,-109.241,-46.226,179.673,4.279,148.796
C00984=1119.488,-109.492,-46.217,179.674,4.274,148.795
C00985=1119.493,-109.742,-46.208,179.675,4.269,148.794
C00986=1119.498,-109.991,-46.199,179.675,4.264,148.793
C00987=1119.504,-110.241,-46.190,179.675,4.259,148.792
C00988=1119.509,-110.490,-46.182,179.675,4.254,148.790
C00989=1119.514,-110.740,-46.173,179.676,4.249,148.789
C00990=1119.520,-110.990,-46.164,179.676,4.243,148.788
C00991=1119.525,-111.240,-46.155,179.676,4.238,148.787
C00992=1119.531,-111.489,-46.146,179.676,4.233,148.786
C00993=1119.536,-111.740,-46.138,179.677,4.228,148.784
C00994=1119.541,-111.989,-46.129,179.677,4.223,148.783
C00995=1119.546,-112.239,-46.120,179.677,4.218,148.782
C00996=1119.552,-112.488,-46.112,179.677,4.212,148.781
C00997=1119.557,-112.738,-46.103,179.678,4.207,148.780
C00998=1119.563,-112.989,-46.095,179.678,4.202,148.778
C00999=1119.568,-113.239,-46.086,179.678,4.197,148.777
C01000=1119.573,-113.454,-46.078,179.678,4.192,148.776
C01001=1119.578,-113.669,-46.071,179.679,4.188,148.775
C01002=1119.583,-113.885,-46.064,179.678,4.183,148.774
C01003=1119.587,-114.100,-46.056,179.679,4.179,148.773
C01004=1119.592,-114.315,-46.048,179.679,4.174,148.772
C01005=1119.596,-114.530,-46.041,179.679,4.170,148.771
C01006=1119.601,-114.746,-46.034,179.679,4.165,148.770
C01007=1119.605,-114.962,-46.026,179.680,4.161,148.769
C01008=1119.611,-115.211,-46.018,179.680,4.156,148.768
C01009=1119.616,-115.461,-46.009,179.681,4.150,148.766
C01010=1119.622,-115.711,-46.001,179.681,4.145,148.765
C01011=1119.627,-115.960,-45.992,179.681,4.140,148.764
C01012=1119.632,-116.210,-45.983,179.681,4.134,148.763
C01013=1119.638,-116.461,-45.975,179.681,4.129,148.762
C01014=1119.643,-116.711,-45.966,179.681,4.124,148.760
C01015=1119.649,-116.960,-45.958,179.682,4.119,148.759
C01016=1119.654,-117.210,-45.950,179.682,4.113,148.758
C01017=1119.659,-117.460,-45.941,179.682,4.108,148.757
C01018=1119.665,-117.709,-45.933,179.683,4.103,148.755
C01019=1119.670,-117.959,-45.924,179.683,4.097,148.754
C01020=1119.676,-118.208,-45.916,179.683,4.092,148.753
C01021=1119.681,-118.459,-45.908,179.683,4.086,148.752
C01022=1119.686,-118.709,-45.899,179.683,4.081,148.750
C01023=1119.692,-118.958,-45.890,179.684,4.076,148.749
C01024=1119.698,-119.208,-45.882,179.684,4.071,148.748
C01025=1119.702,-119.458,-45.874,179.684,4.066,148.747
C01026=1119.708,-119.708,-45.866,179.685,4.060,148.746
C01027=1119.713,-119.958,-45.857,179.685,4.055,148.744
C01028=1119.718,-120.207,-45.848,179.685,4.049,148.743
C01029=1119.725,-120.457,-45.840,179.685,4.044,148.742
C01030=1119.729,-120.707,-45.832,179.686,4.039,148.741
C01031=1119.735,-120.957,-45.824,179.686,4.033,148.739
C01032=1119.740,-121.206,-45.815,179.686,4.028,148.738
C01033=1119.746,-121.457,-45.807,179.686,4.023,148.737
C01034=1119.751,-121.706,-45.799,179.687,4.017,148.735
C01035=1119.756,-121.956,-45.791,179.687,4.011,148.734
C01036=1119.762,-122.205,-45.782,179.687,4.006,148.733
C01037=1119.767,-122.456,-45.774,179.688,4.001,148.732
C01038=1119.773,-122.706,-45.765,179.687,3.995,148.731
C01039=1119.779,-122.955,-45.758,179.688,3.990,148.729
C01040=1119.783,-123.205,-45.749,179.688,3.984,148.728
C01041=1119.789,-123.455,-45.741,179.689,3.979,148.727
C01042=1119.794,-123.705,-45.733,179.689,3.974,148.726
C01043=1119.800,-123.954,-45.725,179.689,3.968,148.724
C01044=1119.805,-124.204,-45.717,179.689,3.963,148.723
C01045=1119.810,-124.454,-45.708,179.690,3.957,148.722
C01046=1119.816,-124.704,-45.700,179.690,3.952,148.720
C01047=1119.821,-124.954,-45.692,179.690,3.946,148.719
C01048=1119.827,-125.203,-45.684,179.690,3.941,148.718
C01049=1119.832,-125.454,-45.676,179.690,3.936,148.717
C01050=1119.837,-125.703,-45.668,179.691,3.929,148.715
C01051=1119.843,-125.953,-45.660,179.691,3.924,148.714
C01052=1119.849,-126.202,-45.651,179.691,3.919,148.713
C01053=1119.854,-126.453,-45.643,179.692,3.914,148.712
C01054=1119.859,-126.702,-45.636,179.692,3.908,148.710
C01055=1119.865,-126.952,-45.627,179.692,3.902,148.709
C01056=1119.869,-127.168,-45.621,179.692,3.898,148.708
C01057=1119.874,-127.383,-45.614,179.692,3.892,148.707
C01058=1119.879,-127.599,-45.607,179.693,3.888,148.706
C01059=1119.883,-127.814,-45.600,179.693,3.883,148.705
C01060=1119.888,-128.029,-45.593,179.693,3.878,148.703
C01061=1119.892,-128.246,-45.586,179.693,3.873,148.702
C01062=1119.897,-128.461,-45.580,179.694,3.869,148.701
C01063=1119.902,-128.676,-45.572,179.694,3.864,148.700
C01064=1119.479,-128.667,-45.598,179.701,3.868,148.699
C01065=1119.474,-128.451,-45.605,179.700,3.873,148.700
C01066=1119.469,-128.236,-45.612,179.701,3.877,148.701
C01067=1119.465,-128.021,-45.619,179.700,3.883,148.702
C01068=1119.460,-127.805,-45.626,179.700,3.888,148.703
C01069=1119.456,-127.589,-45.633,179.700,3.892,148.704
C01070=1119.451,-127.373,-45.640,179.699,3.897,148.706
C01071=1119.446,-127.158,-45.647,179.700,3.902,148.707
C01072=1119.442,-126.943,-45.653,179.699,3.907,148.708
C01073=1119.436,-126.693,-45.661,179.699,3.912,148.709
C01074=1119.431,-126.443,-45.670,179.699,3.917,148.710
C01075=1119.426,-126.193,-45.678,179.698,3.923,148.712
C01076=1119.420,-125.944,-45.686,179.698,3.929,148.713
C01077=1119.415,-125.693,-45.694,179.698,3.934,148.714
C01078=1119.409,-125.444,-45.702,179.698,3.939,148.715
C01079=1119.404,-125.194,-45.711,179.697,3.946,148.717
C01080=1119.398,-124.944,-45.718,179.697,3.951,148.718
C01081=1119.393,-124.695,-45.727,179.697,3.956,148.719
C01082=1119.388,-124.445,-45.735,179.696,3.961,148.720
C01083=1119.382,-124.195,-45.743,179.697,3.967,148.722
C01084=1119.376,-123.945,-45.751,179.696,3.973,148.723
C01085=1119.371,-123.695,-45.759,179.696,3.978,148.724
C01086=1119.367,-123.445,-45.768,179.695,3.983,148.725
C01087=1119.360,-123.196,-45.776,179.696,3.989,148.727
C01088=1119.355,-122.946,-45.784,179.695,3.994,148.728
C01089=1119.349,-122.696,-45.792,179.694,4.000,148.729
C01090=1119.344,-122.446,-45.801,179.694,4.005,148.731
C01091=1119.339,-122.196,-45.809,179.694,4.010,148.732
C01092=1119.334,-121.947,-45.817,179.694,4.016,148.733
C01093=1119.328,-121.696,-45.825,179.694,4.021,148.734
C01094=1119.322,-121.447,-45.834,179.694,4.026,148.735
C01095=1119.317,-121.197,-45.843,179.693,4.032,148.737
C01096=1119.312,-120.947,-45.850,179.693,4.037,148.738
C01097=1119.307,-120.698,-45.859,179.693,4.043,148.739
C01098=1119.301,-120.448,-45.867,179.693,4.048,148.740
C01099=1119.296,-120.198,-45.876,179.692,4.053,148.742
C01100=1119.290,-119.948,-45.884,179.692,4.059,148.743
C01101=1119.285,-119.698,-45.893,179.692,4.064,148.744
C01102=1119.280,-119.449,-45.901,179.691,4.069,148.746
C01103=1119.274,-119.199,-45.909,179.691,4.075,148.747
C01104=1119.269,-118.949,-45.918,179.691,4.081,148.748
C01105=1119.263,-118.700,-45.926,179.691,4.086,148.749
C01106=1119.258,-118.449,-45.935,179.690,4.091,148.750
C01107=1119.253,-118.200,-45.943,179.690,4.096,148.752
C01108=1119.247,-117.950,-45.951,179.690,4.101,148.753
C01109=1119.241,-117.700,-45.960,179.690,4.106,148.754
C01110=1119.236,-117.450,-45.969,179.689,4.112,148.755
C01111=1119.231,-117.201,-45.977,179.689,4.117,148.756
C01112=1119.226,-116.951,-45.985,179.688,4.122,148.758
C01113=1119.221,-116.701,-45.994,179.688,4.128,148.759
C01114=1119.215,-116.451,-46.003,179.688,4.133,148.760
C01115=1119.209,-116.201,-46.011,179.688,4.139,148.761
C01116=1119.204,-115.951,-46.020,179.688,4.144,148.763
C01117=1119.199,-115.702,-46.029,179.687,4.149,148.764
C01118=1119.193,-115.452,-46.037,179.687,4.154,148.765
C01119=1119.188,-115.202,-46.045,179.687,4.159,148.766
C01120=1119.183,-114.952,-46.054,179.687,4.164,148.768
C01121=1119.178,-114.737,-46.062,179.687,4.169,148.768
C01122=1119.173,-114.521,-46.069,179.686,4.174,148.770
C01123=1119.168,-114.306,-46.077,179.686,4.178,148.771
C01124=1119.164,-114.091,-46.084,179.686,4.182,148.772
C01125=1119.160,-113.876,-46.091,179.685,4.187,148.773
C01126=1119.154,-113.660,-46.098,179.685,4.192,148.774
C01127=1119.150,-113.444,-46.106,179.685,4.196,148.775
C01128=1119.145,-113.229,-46.114,179.685,4.201,148.776
C01129=1119.140,-112.979,-46.123,179.685,4.206,148.777
C01130=1119.134,-112.730,-46.131,179.684,4.211,148.778
C01131=1119.129,-112.480,-46.140,179.684,4.216,148.780
C01132=1119.124,-112.230,-46.148,179.684,4.221,148.781
C01133=1119.119,-111.980,-46.157,179.683,4.227,148.782
C01134=1119.113,-111.731,-46.166,179.683,4.232,148.783
C01135=1119.108,-111.481,-46.175,179.683,4.237,148.784
C01136=1119.103,-111.231,-46.184,179.683,4.242,148.786
C01137=1119.097,-110.981,-46.192,179.682,4.247,148.787
C01138=1119.092,-110.731,-46.201,179.682,4.252,148.788
C01139=1119.086,-110.482,-46.210,179.682,4.258,148.789
C01140=1119.080,-110.231,-46.219,179.682,4.263,148.790
C01141=1119.075,-109.982,-46.228,179.681,4.268,148.792
C01142=1119.070,-109.732,-46.236,179.681,4.273,148.793
C01143=1119.065,-109.482,-46.245,179.681,4.278,148.794
C01144=1119.059,-109.233,-46.254,179.681,4.283,148.795
C01145=1119.054,-108.983,-46.263,179.680,4.289,148.796
C01146=1119.049,-108.733,-46.272,179.680,4.293,148.798
C01147=1119.044,-108.483,-46.281,179.679,4.298,148.799
C01148=1119.038,-108.233,-46.289,179.679,4.303,148.800
C01149=1119.032,-107.983,-46.299,179.679,4.308,148.801
C01150=1119.027,-107.734,-46.308,179.679,4.314,148.802
C01151=1119.022,-107.484,-46.316,179.678,4.319,148.804
C01152=1119.016,-107.234,-46.325,179.678,4.324,148.805
C01153=1119.011,-106.984,-46.334,179.678,4.329,148.806
C01154=1119.006,-106.735,-46.343,179.678,4.334,148.807
C01155=1119.001,-106.485,-46.352,179.677,4.339,148.808
C01156=1118.995,-106.235,-46.361,179.677,4.345,148.810
C01157=1118.989,-105.985,-46.370,179.677,4.350,148.811
C01158=1118.984,-105.736,-46.379,179.676,4.354,148.812
C01159=1118.979,-105.486,-46.388,179.676,4.359,148.813
C01160=1118.974,-105.236,-46.397,179.676,4.364,148.814
C01161=1118.969,-104.987,-46.406,179.675,4.370,148.816
C01162=1118.963,-104.736,-46.416,179.676,4.374,148.816
C01163=1118.958,-104.487,-46.425,179.675,4.380,148.818
C01164=1118.953,-104.237,-46.434,179.675,4.385,148.819
C01165=1118.947,-103.987,-46.443,179.675,4.390,148.820
C01166=1118.942,-103.738,-46.451,179.674,4.394,148.821
C01167=1118.936,-103.488,-46.461,179.674,4.399,148.822
C01168=1118.931,-103.238,-46.469,179.674,4.405,148.824
C01169=1118.925,-102.988,-46.478,179.673,4.410,148.825
C01170=1118.921,-102.739,-46.488,179.673,4.415,148.826
C01171=1118.915,-102.488,-46.497,179.673,4.420,148.827
C01172=1118.909,-102.239,-46.506,179.673,4.425,148.828
C01173=1118.904,-101.989,-46.515,179.672,4.430,148.830
C01174=1118.899,-101.739,-46.524,179.672,4.435,148.831
C01175=1118.894,-101.489,-46.534,179.672,4.440,148.832
C01176=1118.888,-101.240,-46.543,179.671,4.445,148.833
C01177=1118.884,-101.024,-46.551,179.671,4.449,148.834
C01178=1118.879,-100.809,-46.559,179.671,4.453,148.835
C01179=1118.875,-100.594,-46.566,179.671,4.458,148.836
C01180=1118.870,-100.378,-46.574,179.670,4.462,148.837
C01181=1118.865,-100.162,-46.583,179.670,4.466,148.838
C01182=1118.860,-99.948,-46.591,179.670,4.471,148.839
C01183=1118.856,-99.732,-46.599,179.669,4.475,148.840
C01184=1118.851,-99.517,-46.607,179.669,4.479,148.841
C01185=1118.846,-99.267,-46.615,179.669,4.484,148.842
C01186=1118.840,-99.018,-46.626,179.669,4.489,148.844
C01187=1118.835,-98.768,-46.635,179.668,4.494,148.845
C01188=1118.830,-98.518,-46.643,179.668,4.499,148.846
C01189=1118.824,-98.268,-46.653,179.668,4.504,148.847
C01190=1118.819,-98.018,-46.663,179.668,4.509,148.848
C01191=1118.814,-97.769,-46.671,179.668,4.514,148.849
C01192=1118.808,-97.518,-46.681,179.667,4.518,148.851
C01193=1118.803,-97.269,-46.691,179.666,4.524,148.852
C01194=1118.798,-97.019,-46.700,179.666,4.529,148.853
C01195=1118.792,-96.769,-46.709,179.666,4.534,148.854
C01196=1118.788,-96.520,-46.719,179.665,4.538,148.855
C01197=1118.782,-96.270,-46.728,179.665,4.543,148.857
C01198=1118.776,-96.020,-46.737,179.665,4.549,148.858
C01199=1118.771,-95.770,-46.747,179.665,4.554,148.859
C01200=1118.766,-95.521,-46.756,179.664,4.558,148.860
C01201=1118.761,-95.271,-46.765,179.664,4.563,148.861
C01202=1118.755,-95.021,-46.775,179.663,4.568,148.862
C01203=1118.750,-94.771,-46.784,179.663,4.574,148.864
C01204=1118.744,-94.522,-46.794,179.662,4.578,148.865
C01205=1118.739,-94.272,-46.803,179.662,4.583,148.866
C01206=1118.734,-94.022,-46.812,179.661,4.587,148.867
C01207=1118.728,-93.773,-46.822,179.661,4.593,148.868
C01208=1118.723,-93.523,-46.831,179.660,4.597,148.870
C01209=1118.717,-93.273,-46.841,179.660,4.602,148.871
C01210=1118.712,-93.023,-46.850,179.659,4.607,148.872
C01211=1118.707,-92.774,-46.861,179.658,4.611,148.873
C01212=1118.702,-92.524,-46.869,179.658,4.616,148.875
C01213=1118.696,-92.273,-46.879,179.657,4.621,148.876
C01214=1118.691,-92.024,-46.889,179.657,4.626,148.877
C01215=1118.685,-91.774,-46.898,179.656,4.630,148.878
C01216=1118.681,-91.524,-46.908,179.655,4.636,148.880
C01217=1118.675,-91.274,-46.917,179.655,4.640,148.881
C01218=1118.670,-91.025,-46.927,179.655,4.645,148.882
C01219=1118.664,-90.775,-46.937,179.654,4.650,148.883
C01220=1118.659,-90.526,-46.946,179.654,4.655,148.884
C01221=1118.653,-90.275,-46.956,179.653,4.660,148.886
C01222=1118.648,-90.026,-46.965,179.652,4.665,148.887
C01223=1118.642,-89.776,-46.975,179.652,4.670,148.888
C01224=1118.638,-89.526,-46.985,179.651,4.674,148.889
C01225=1118.633,-89.277,-46.995,179.651,4.679,148.890
C01226=1118.627,-89.027,-47.004,179.650,4.685,148.892
C01227=1118.622,-88.777,-47.014,179.649,4.689,148.893
C01228=1118.617,-88.527,-47.023,179.649,4.694,148.894
C01229=1118.611,-88.278,-47.033,179.649,4.700,148.895
C01230=1118.606,-88.028,-47.042,179.648,4.704,148.897
C01231=1118.600,-87.778,-47.052,179.648,4.709,148.898
C01232=1118.596,-87.528,-47.062,179.647,4.715,148.899
C01233=1118.590,-87.313,-47.070,179.647,4.719,148.900
C01234=1118.587,-87.098,-47.079,179.646,4.723,148.901
C01235=1118.582,-86.883,-47.087,179.646,4.727,148.902
C01236=1118.577,-86.667,-47.096,179.646,4.731,148.903
C01237=1118.572,-86.452,-47.104,179.646,4.736,148.904
C01238=1118.568,-86.237,-47.112,179.645,4.740,148.905
C01239=1118.563,-86.022,-47.121,179.645,4.744,148.906
C01240=1118.559,-85.806,-47.129,179.644,4.748,148.907
C01241=1118.553,-85.557,-47.140,179.644,4.753,148.909
C01242=1118.548,-85.307,-47.148,179.644,4.759,148.910
C01243=1118.543,-85.058,-47.159,179.643,4.764,148.911
C01244=1118.538,-84.807,-47.169,179.643,4.768,148.912
C01245=1118.532,-84.557,-47.178,179.642,4.774,148.914
C01246=1118.527,-84.308,-47.188,179.642,4.779,148.915
C01247=1118.522,-84.059,-47.198,179.642,4.784,148.916
C01248=1118.516,-83.808,-47.207,179.642,4.789,148.917
C01249=1118.510,-83.559,-47.218,179.642,4.794,148.918
C01250=1118.506,-83.309,-47.228,179.641,4.799,148.919
C01251=1118.500,-83.059,-47.237,179.640,4.804,148.921
C01252=1118.495,-82.809,-47.247,179.640,4.809,148.922
C01253=1118.490,-82.560,-47.257,179.640,4.814,148.923
C01254=1118.484,-82.311,-47.267,179.640,4.820,148.924
C01255=1118.479,-82.060,-47.277,179.640,4.825,148.926
C01256=1118.474,-81.810,-47.287,179.639,4.830,148.927
C01257=1118.468,-81.561,-47.297,179.639,4.835,148.928
C01258=1118.463,-81.311,-47.307,179.639,4.840,148.929
C01259=1118.458,-81.061,-47.318,179.639,4.845,148.930
C01260=1118.453,-80.811,-47.326,179.639,4.851,148.931
C01261=1118.447,-80.562,-47.337,179.639,4.856,148.933
C01262=1118.441,-80.312,-47.347,179.638,4.860,148.934
C01263=1118.437,-80.062,-47.357,179.638,4.865,148.935
C01264=1118.432,-79.813,-47.367,179.637,4.870,148.936
C01265=1118.426,-79.563,-47.377,179.637,4.876,148.937
C01266=1118.420,-79.313,-47.387,179.637,4.881,148.938
C01267=1118.416,-79.063,-47.397,179.637,4.886,148.940
C01268=1118.410,-78.813,-47.407,179.637,4.891,148.941
C01269=1118.405,-78.564,-47.417,179.637,4.897,148.942
C01270=1118.399,-78.314,-47.427,179.637,4.902,148.943
C01271=1118.394,-78.064,-47.438,179.637,4.907,148.944
C01272=1118.389,-77.815,-47.448,179.637,4.912,148.945
C01273=1118.383,-77.565,-47.457,179.637,4.918,148.947
C01274=1118.378,-77.315,-47.467,179.637,4.923,148.948
C01275=1118.373,-77.065,-47.478,179.636,4.928,148.949
C01276=1118.367,-76.815,-47.488,179.636,4.933,148.950
C01277=1118.361,-76.566,-47.498,179.636,4.938,148.951
C01278=1118.357,-76.316,-47.508,179.636,4.943,148.952
C01279=1118.352,-76.066,-47.518,179.636,4.948,148.954
C01280=1118.346,-75.817,-47.529,179.636,4.954,148.955
C01281=1118.341,-75.567,-47.539,179.636,4.958,148.956
C01282=1118.335,-75.317,-47.549,179.636,4.964,148.957
C01283=1118.330,-75.068,-47.560,179.636,4.969,148.958
C01284=1118.326,-74.818,-47.570,179.636,4.975,148.959
C01285=1118.320,-74.568,-47.580,179.636,4.980,148.960
C01286=1118.314,-74.319,-47.590,179.636,4.985,148.962
C01287=1118.309,-74.068,-47.601,179.636,4.990,148.963
C01288=1118.304,-73.819,-47.611,179.637,4.996,148.964
C01289=1118.299,-73.603,-47.620,179.636,5.000,148.965
C01290=1118.295,-73.389,-47.628,179.636,5.005,148.966
C01291=1118.290,-73.173,-47.638,179.636,5.009,148.967
C01292=1118.286,-72.958,-47.646,179.636,5.013,148.968
C01293=1118.281,-72.743,-47.655,179.637,5.018,148.969
C01294=1118.276,-72.528,-47.665,179.636,5.022,148.969
C01295=1118.272,-72.313,-47.673,179.637,5.027,148.970
C01296=1118.267,-72.098,-47.682,179.637,5.032,148.971
C01297=1118.262,-71.848,-47.693,179.637,5.037,148.972
C01298=1118.256,-71.598,-47.703,179.637,5.042,148.974
C01299=1118.251,-71.349,-47.713,179.637,5.047,148.975
C01300=1118.246,-71.098,-47.724,179.638,5.053,148.976
C01301=1118.240,-70.849,-47.734,179.638,5.058,148.977
C01302=1118.236,-70.599,-47.745,179.638,5.063,148.978
C01303=1118.230,-70.350,-47.756,179.638,5.068,148.979
C01304=1118.225,-70.099,-47.766,179.638,5.074,148.980
C01305=1118.219,-69.850,-47.776,179.639,5.079,148.981
C01306=1118.214,-69.600,-47.787,179.639,5.084,148.982
C01307=1118.209,-69.351,-47.798,179.639,5.088,148.983
C01308=1118.203,-69.101,-47.808,179.639,5.094,148.984
C01309=1118.198,-68.851,-47.819,179.639,5.100,148.985
C01310=1118.193,-68.601,-47.829,179.640,5.104,148.986
C01311=1118.188,-68.351,-47.839,179.640,5.110,148.988
C01312=1118.183,-68.102,-47.850,179.640,5.115,148.988
C01313=1118.178,-67.852,-47.861,179.640,5.120,148.990
C01314=1118.172,-67.602,-47.871,179.641,5.126,148.991
C01315=1118.167,-67.353,-47.882,179.641,5.131,148.992
C01316=1118.162,-67.103,-47.893,179.642,5.136,148.993
C01317=1118.156,-66.854,-47.903,179.642,5.142,148.994
C01318=1118.151,-66.603,-47.913,179.642,5.146,148.995
C01319=1118.146,-66.354,-47.924,179.642,5.152,148.996
C01320=1118.141,-66.104,-47.935,179.643,5.157,148.997
C01321=1118.135,-65.855,-47.945,179.644,5.162,148.998
C01322=1118.131,-65.605,-47.956,179.644,5.168,148.999
C01323=1118.124,-65.355,-47.967,179.644,5.173,149.000
C01324=1118.119,-65.106,-47.978,179.645,5.177,149.001
C01325=1118.114,-64.855,-47.989,179.645,5.183,149.002
C01326=1118.109,-64.606,-47.999,179.646,5.188,149.003
C01327=1118.104,-64.356,-48.011,179.647,5.194,149.004
C01328=1118.099,-64.107,-48.021,179.647,5.199,149.005
C01329=1118.094,-63.857,-48.032,179.647,5.203,149.006
C01330=1118.088,-63.607,-48.043,179.648,5.209,149.007
C01331=1118.083,-63.357,-48.053,179.648,5.214,149.008
C01332=1118.077,-63.108,-48.064,179.649,5.220,149.009
C01333=1118.072,-62.858,-48.075,179.649,5.225,149.010
C01334=1118.067,-62.609,-48.086,179.650,5.230,149.011
C01335=1118.062,-62.359,-48.096,179.651,5.235,149.012
C01336=1118.057,-62.109,-48.108,179.652,5.240,149.012
C01337=1118.051,-61.859,-48.119,179.652,5.245,149.013
C01338=1118.046,-61.609,-48.130,179.652,5.250,149.015
C01339=1118.041,-61.360,-48.140,179.653,5.256,149.015
C01340=1118.035,-61.110,-48.152,179.653,5.261,149.016
C01341=1118.031,-60.860,-48.163,179.654,5.266,149.017
C01342=1118.025,-60.611,-48.173,179.655,5.271,149.018
C01343=1118.020,-60.361,-48.185,179.656,5.276,149.019
C01344=1118.015,-60.111,-48.196,179.656,5.281,149.020
C01345=1118.010,-59.897,-48.205,179.656,5.285,149.021
C01346=1118.006,-59.681,-48.214,179.656,5.289,149.022
C01347=1118.001,-59.466,-48.224,179.656,5.294,149.023
C01348=1117.997,-59.251,-48.233,179.656,5.298,149.024
C01349=1117.992,-59.036,-48.243,179.656,5.302,149.025
C01350=1117.988,-58.821,-48.253,179.655,5.306,149.026
C01351=1117.983,-58.606,-48.263,179.655,5.310,149.026
C01352=1117.978,-58.391,-48.272,179.655,5.314,149.027
C01353=1117.973,-58.141,-48.283,179.655,5.318,149.028
C01354=1117.968,-57.891,-48.294,179.655,5.323,149.029
C01355=1117.962,-57.642,-48.305,179.655,5.328,149.030
C01356=1117.958,-57.392,-48.316,179.654,5.332,149.032
C01357=1117.953,-57.142,-48.327,179.654,5.337,149.033
C01358=1117.947,-56.893,-48.338,179.655,5.342,149.034
C01359=1117.942,-56.643,-48.350,179.654,5.346,149.035
C01360=1117.937,-56.393,-48.360,179.654,5.351,149.036
C01361=1117.932,-56.143,-48.372,179.654,5.355,149.037
C01362=1117.926,-55.894,-48.383,179.654,5.360,149.038
C01363=1117.922,-55.644,-48.394,179.654,5.365,149.039
C01364=1117.916,-55.394,-48.406,179.653,5.369,149.040
C01365=1117.911,-55.145,-48.417,179.653,5.375,149.041
C01366=1117.905,-54.895,-48.428,179.653,5.379,149.042
C01367=1117.900,-54.645,-48.440,179.653,5.384,149.043
C01368=1117.895,-54.396,-48.450,179.653,5.389,149.044
C01369=1117.889,-54.146,-48.462,179.652,5.393,149.046
C01370=1117.885,-53.896,-48.473,179.653,5.398,149.047
C01371=1117.879,-53.646,-48.485,179.652,5.402,149.048
C01372=1117.874,-53.397,-48.495,179.652,5.407,149.049
C01373=1117.869,-53.147,-48.506,179.652,5.412,149.050
C01374=1117.864,-52.897,-48.518,179.652,5.416,149.051
C01375=1117.859,-52.648,-48.530,179.651,5.422,149.052
C01376=1117.853,-52.398,-48.541,179.651,5.426,149.053
C01377=1117.848,-52.149,-48.552,179.651,5.431,149.054
C01378=1117.842,-51.898,-48.564,179.651,5.436,149.055
C01379=1117.838,-51.648,-48.575,179.651,5.440,149.056
C01380=1117.832,-51.400,-48.586,179.651,5.445,149.057
C01381=1117.827,-51.150,-48.598,179.650,5.449,149.058
C01382=1117.822,-50.900,-48.609,179.651,5.454,149.059
C01383=1117.817,-50.650,-48.621,179.650,5.459,149.061
C01384=1117.812,-50.401,-48.632,179.650,5.463,149.062
C01385=1117.806,-50.151,-48.643,179.650,5.468,149.063
C01386=1117.801,-49.901,-48.654,179.650,5.473,149.064
C01387=1117.796,-49.651,-48.666,179.649,5.478,149.065
C01388=1117.790,-49.402,-48.677,179.649,5.483,149.066
C01389=1117.785,-49.152,-48.689,179.649,5.487,149.067
C01390=1117.780,-48.903,-48.700,179.649,5.492,149.068
C01391=1117.775,-48.653,-48.712,179.648,5.496,149.069
C01392=1117.770,-48.404,-48.723,179.649,5.501,149.070
C01393=1117.764,-48.154,-48.735,179.649,5.506,149.071
C01394=1117.759,-47.904,-48.747,179.648,5.510,149.072
C01395=1117.754,-47.654,-48.758,179.648,5.516,149.074
C01396=1117.749,-47.404,-48.770,179.648,5.520,149.074
C01397=1117.744,-47.155,-48.781,179.648,5.525,149.076
C01398=1117.738,-46.905,-48.793,179.648,5.530,149.077
C01399=1117.733,-46.656,-48.804,179.648,5.534,149.078
C01400=1117.728,-46.406,-48.816,179.648,5.539,149.079
C01401=1117.723,-46.190,-48.825,179.647,5.543,149.080
C01402=1117.719,-45.975,-48.835,179.647,5.547,149.081
C01403=1117.714,-45.761,-48.845,179.647,5.551,149.082
C01404=1117.710,-45.546,-48.855,179.647,5.555,149.083
C01405=1117.705,-45.331,-48.866,179.647,5.559,149.083
C01406=1117.701,-45.116,-48.876,179.646,5.563,149.085
C01407=1117.696,-44.901,-48.886,179.646,5.567,149.085
C01408=1117.692,-44.686,-48.896,179.646,5.572,149.086
C01409=1117.687,-44.436,-48.908,179.646,5.576,149.087
C01410=1117.682,-44.186,-48.919,179.646,5.581,149.088
C01411=1117.676,-43.937,-48.931,179.645,5.585,149.090
C01412=1117.671,-43.688,-48.942,179.645,5.590,149.091
C01413=1117.666,-43.438,-48.954,179.646,5.595,149.092
C01414=1117.660,-43.188,-48.966,179.645,5.599,149.093
C01415=1117.656,-42.938,-48.977,179.645,5.604,149.094
C01416=1117.650,-42.688,-48.989,179.647,5.610,149.095
C01417=1117.645,-42.438,-49.001,179.648,5.615,149.095
C01418=1117.640,-42.189,-49.012,179.649,5.621,149.096
C01419=1117.635,-41.939,-49.025,179.650,5.626,149.097
C01420=1117.629,-41.690,-49.036,179.651,5.631,149.098
C01421=1117.624,-41.440,-49.047,179.652,5.637,149.099
C01422=1117.619,-41.190,-49.059,179.654,5.642,149.100
C01423=1117.613,-40.940,-49.071,179.655,5.648,149.100
C01424=1117.608,-40.691,-49.084,179.655,5.652,149.101
C01425=1117.604,-40.442,-49.095,179.657,5.657,149.102
C01426=1117.598,-40.192,-49.107,179.658,5.663,149.103
C01427=1117.593,-39.942,-49.119,179.659,5.668,149.104
C01428=1117.588,-39.692,-49.131,179.660,5.673,149.105
C01429=1117.583,-39.443,-49.143,179.661,5.678,149.105
C01430=1117.577,-39.193,-49.155,179.662,5.683,149.106
C01431=1117.572,-38.943,-49.167,179.663,5.688,149.107
C01432=1117.567,-38.694,-49.179,179.663,5.693,149.108
C01433=1117.562,-38.444,-49.190,179.665,5.698,149.109
C01434=1117.557,-38.194,-49.202,179.665,5.703,149.109
C01435=1117.552,-37.945,-49.215,179.666,5.707,149.110
C01436=1117.546,-37.695,-49.227,179.667,5.713,149.111
C01437=1117.541,-37.445,-49.239,179.668,5.718,149.112
C01438=1117.536,-37.195,-49.251,179.669,5.722,149.113
C01439=1117.531,-36.946,-49.263,179.669,5.727,149.114
C01440=1117.526,-36.696,-49.275,179.670,5.732,149.114
C01441=1117.520,-36.447,-49.287,179.671,5.737,149.115
C01442=1117.515,-36.197,-49.299,179.671,5.741,149.116
C01443=1117.510,-35.947,-49.312,179.672,5.746,149.117
C01444=1117.504,-35.697,-49.323,179.673,5.750,149.118
C01445=1117.499,-35.448,-49.336,179.673,5.755,149.118
C01446=1117.495,-35.198,-49.347,179.674,5.760,149.119
C01447=1117.489,-34.949,-49.360,179.674,5.765,149.120
C01448=1117.484,-34.699,-49.372,179.675,5.769,149.121
C01449=1117.479,-34.449,-49.384,179.676,5.774,149.122
C01450=1117.474,-34.200,-49.396,179.675,5.778,149.123
C01451=1117.468,-33.950,-49.408,179.676,5.782,149.124
C01452=1117.463,-33.701,-49.421,179.676,5.787,149.125
C01453=1117.458,-33.451,-49.433,179.677,5.792,149.125
C01454=1117.452,-33.201,-49.445,179.677,5.796,149.126
C01455=1117.447,-32.952,-49.458,179.678,5.800,149.127
C01456=1117.442,-32.702,-49.470,179.678,5.805,149.128
C01457=1117.438,-32.487,-49.480,179.678,5.809,149.129
C01458=1117.433,-32.272,-49.491,179.678,5.812,149.130
C01459=1117.429,-32.057,-49.501,179.679,5.816,149.130
C01460=1117.425,-31.843,-49.512,179.678,5.820,149.131
C01461=1117.420,-31.628,-49.523,179.679,5.824,149.132
C01462=1117.416,-31.413,-49.533,179.679,5.827,149.133
C01463=1117.411,-31.198,-49.544,179.679,5.831,149.133
C01464=1117.407,-30.983,-49.554,179.679,5.835,149.134
C01465=1117.402,-30.733,-49.567,179.679,5.839,149.135
C01466=1117.396,-30.483,-49.579,179.679,5.844,149.136
C01467=1117.391,-30.234,-49.592,179.679,5.848,149.137
C01468=1117.386,-29.985,-49.604,179.680,5.852,149.138
C01469=1117.381,-29.735,-49.616,179.679,5.857,149.139
C01470=1117.376,-29.485,-49.629,179.679,5.861,149.140
C01471=1117.371,-29.235,-49.641,179.679,5.865,149.141
C01472=1117.366,-28.986,-49.653,179.679,5.869,149.142
C01473=1117.361,-28.736,-49.666,179.678,5.874,149.143
C01474=1117.355,-28.486,-49.678,179.678,5.878,149.144
C01475=1117.350,-28.237,-49.691,179.678,5.882,149.145
C01476=1117.344,-27.987,-49.704,179.678,5.886,149.146
C01477=1117.339,-27.737,-49.716,179.677,5.890,149.147
C01478=1117.334,-27.487,-49.729,179.677,5.894,149.148
C01479=1117.329,-27.238,-49.741,179.677,5.899,149.149
C01480=1117.324,-26.989,-49.754,179.677,5.903,149.150
C01481=1117.319,-26.739,-49.766,179.676,5.907,149.151
C01482=1117.313,-26.490,-49.778,179.675,5.912,149.152
C01483=1117.309,-26.240,-49.791,179.675,5.916,149.153
C01484=1117.303,-25.990,-49.803,179.674,5.919,149.154
C01485=1117.298,-25.740,-49.816,179.674,5.924,149.155
C01486=1117.293,-25.491,-49.828,179.675,5.929,149.156
C01487=1117.288,-25.242,-49.841,179.675,5.934,149.157
C01488=1117.283,-24.991,-49.853,179.675,5.939,149.158
C01489=1117.278,-24.742,-49.866,179.677,5.944,149.159
C01490=1117.272,-24.492,-49.879,179.677,5.949,149.160
C01491=1117.267,-24.243,-49.892,179.678,5.954,149.161
C01492=1117.262,-23.993,-49.904,179.678,5.958,149.162
C01493=1117.257,-23.743,-49.916,179.678,5.963,149.163
C01494=1117.252,-23.494,-49.929,179.679,5.968,149.163
C01495=1117.247,-23.244,-49.942,179.679,5.973,149.164
C01496=1117.241,-22.995,-49.955,179.680,5.977,149.165
C01497=1117.236,-22.745,-49.967,179.680,5.982,149.166
C01498=1117.231,-22.495,-49.980,179.682,5.987,149.167
C01499=1117.226,-22.245,-49.992,179.682,5.992,149.168
C01500=1117.221,-21.996,-50.005,179.683,5.997,149.169
C01501=1117.216,-21.747,-50.018,179.683,6.001,149.169
C01502=1117.211,-21.496,-50.031,179.684,6.006,149.170
C01503=1117.205,-21.247,-50.044,179.684,6.011,149.171
C01504=1117.200,-20.998,-50.056,179.685,6.016,149.172
C01505=1117.195,-20.748,-50.069,179.685,6.020,149.173
C01506=1117.190,-20.498,-50.082,179.686,6.025,149.174
C01507=1117.185,-20.249,-50.095,179.687,6.029,149.175
C01508=1117.180,-19.999,-50.108,179.687,6.034,149.176
C01509=1117.175,-19.750,-50.120,179.688,6.039,149.176
C01510=1117.169,-19.500,-50.134,179.688,6.044,149.177
C01511=1117.164,-19.250,-50.146,179.689,6.049,149.178
C01512=1117.159,-19.001,-50.159,179.690,6.054,149.179
C01513=1117.155,-18.785,-50.170,179.690,6.057,149.180
C01514=1117.150,-18.571,-50.181,179.691,6.062,149.180
C01515=1117.146,-18.356,-50.192,179.691,6.066,149.181
C01516=1117.142,-18.141,-50.204,179.691,6.069,149.182
C01517=1117.137,-17.927,-50.215,179.692,6.073,149.183
C01518=1117.132,-17.712,-50.225,179.693,6.077,149.183
C01519=1117.128,-17.497,-50.237,179.693,6.082,149.184
C01520=1117.124,-17.282,-50.248,179.694,6.085,149.185
C01521=1117.118,-17.033,-50.261,179.694,6.090,149.186
C01522=1117.113,-16.782,-50.274,179.695,6.095,149.187
C01523=1117.108,-16.533,-50.287,179.696,6.099,149.187
C01524=1117.103,-16.284,-50.299,179.696,6.104,149.188
C01525=1117.098,-16.033,-50.313,179.697,6.109,149.189
C01526=1117.093,-15.785,-50.326,179.697,6.113,149.190
C01527=1117.088,-15.535,-50.339,179.698,6.118,149.191
C01528=1117.082,-15.285,-50.352,179.698,6.122,149.192
C01529=1117.077,-15.036,-50.365,179.699,6.127,149.193
C01530=1117.073,-14.786,-50.378,179.699,6.132,149.193
C01531=1117.067,-14.536,-50.391,179.700,6.136,149.194
C01532=1117.062,-14.287,-50.404,179.701,6.141,149.195
C01533=1117.057,-14.037,-50.418,179.701,6.146,149.196
C01534=1117.052,-13.788,-50.431,179.702,6.150,149.197
C01535=1117.047,-13.538,-50.444,179.703,6.155,149.197
C01536=1117.041,-13.288,-50.457,179.703,6.159,149.198
C01537=1117.037,-13.039,-50.470,179.704,6.164,149.199
C01538=1117.031,-12.789,-50.484,179.704,6.169,149.200
C01539=1117.026,-12.540,-50.496,179.705,6.173,149.201
C01540=1117.021,-12.289,-50.510,179.706,6.178,149.202
C01541=1117.016,-12.041,-50.523,179.706,6.183,149.203
C01542=1117.010,-11.791,-50.536,179.707,6.187,149.203
C01543=1117.006,-11.541,-50.549,179.708,6.192,149.204
C01544=1117.001,-11.292,-50.562,179.708,6.196,149.205
C01545=1116.996,-11.042,-50.576,179.709,6.201,149.206
C01546=1116.990,-10.793,-50.589,179.710,6.206,149.207
C01547=1116.985,-10.542,-50.602,179.710,6.210,149.207
C01548=1116.980,-10.294,-50.616,179.711,6.215,149.208
C01549=1116.975,-10.043,-50.629,179.711,6.220,149.209
C01550=1116.970,-9.794,-50.642,179.712,6.223,149.210
C01551=1116.965,-9.544,-50.656,179.712,6.228,149.211
C01552=1116.959,-9.295,-50.669,179.713,6.233,149.212
C01553=1116.955,-9.045,-50.683,179.714,6.237,149.212
C01554=1116.949,-8.796,-50.696,179.714,6.242,149.213
C01555=1116.945,-8.546,-50.709,179.715,6.246,149.214
C01556=1116.939,-8.297,-50.723,179.715,6.251,149.215
C01557=1116.935,-8.047,-50.736,179.716,6.256,149.216
C01558=1116.929,-7.798,-50.750,179.717,6.260,149.217
C01559=1116.924,-7.548,-50.763,179.717,6.265,149.217
C01560=1116.919,-7.299,-50.777,179.718,6.269,149.218
C01561=1116.914,-7.048,-50.790,179.719,6.274,149.219
C01562=1116.908,-6.799,-50.803,179.719,6.279,149.220
C01563=1116.904,-6.549,-50.817,179.720,6.282,149.221
C01564=1116.898,-6.300,-50.830,179.720,6.287,149.221
C01565=1116.893,-6.050,-50.844,179.721,6.292,149.222
C01566=1116.888,-5.801,-50.857,179.721,6.296,149.223
C01567=1116.883,-5.551,-50.871,179.722,6.301,149.224
C01568=1116.878,-5.302,-50.884,179.723,6.306,149.225
C01569=1116.874,-5.087,-50.897,179.723,6.309,149.225
C01570=1116.869,-4.872,-50.908,179.724,6.313,149.226
C01571=1116.865,-4.657,-50.920,179.725,6.317,149.227
C01572=1116.860,-4.443,-50.932,179.724,6.321,149.228
C01573=1116.856,-4.228,-50.943,179.725,6.325,149.228
C01574=1116.851,-4.013,-50.955,179.726,6.329,149.229
C01575=1116.847,-3.798,-50.966,179.726,6.332,149.230
C01576=1116.843,-3.584,-50.978,179.727,6.337,149.230
C01577=1116.837,-3.334,-50.992,179.728,6.341,149.231
C01578=1116.833,-3.084,-51.006,179.728,6.346,149.232
C01579=1116.828,-2.835,-51.020,179.729,6.350,149.233
C01580=1116.822,-2.585,-51.033,179.729,6.354,149.234
C01581=1116.817,-2.336,-51.047,179.730,6.359,149.235
C01582=1116.812,-2.086,-51.060,179.730,6.364,149.235
C01583=1116.807,-1.836,-51.074,179.731,6.368,149.236
C01584=1116.802,-1.587,-51.088,179.732,6.373,149.237
C01585=1116.797,-1.337,-51.102,179.732,6.378,149.238
C01586=1116.792,-1.088,-51.115,179.733,6.382,149.239
C01587=1116.787,-0.839,-51.129,179.734,6.387,149.239
C01588=1116.781,-0.588,-51.143,179.734,6.391,149.240
C01589=1116.776,-0.339,-51.157,179.734,6.395,149.241
C01590=1116.772,-0.090,-51.170,179.735,6.400,149.242
C01591=1116.767,0.160,-51.185,179.736,6.404,149.243
C01592=1116.761,0.410,-51.198,179.736,6.409,149.244
C01593=1116.756,0.659,-51.212,179.737,6.414,149.245
C01594=1116.751,0.909,-51.226,179.738,6.418,149.245
C01595=1116.746,1.158,-51.240,179.738,6.423,149.246
C01596=1116.741,1.408,-51.253,179.739,6.427,149.247
C01597=1116.736,1.658,-51.268,179.739,6.431,149.248
C01598=1116.730,1.907,-51.282,179.740,6.436,149.249
C01599=1116.725,2.156,-51.296,179.740,6.440,149.249
C01600=1116.721,2.406,-51.310,179.741,6.445,149.250
C01601=1116.715,2.655,-51.323,179.741,6.450,149.251
C01602=1116.710,2.905,-51.337,179.742,6.454,149.252
C01603=1116.705,3.155,-51.351,179.743,6.459,149.253
C01604=1116.700,3.404,-51.365,179.744,6.464,149.254
C01605=1116.695,3.654,-51.379,179.743,6.468,149.254
C01606=1116.690,3.903,-51.394,179.744,6.472,149.255
C01607=1116.685,4.153,-51.408,179.745,6.477,149.256
C01608=1116.679,4.403,-51.421,179.746,6.481,149.257
C01609=1116.675,4.652,-51.435,179.746,6.486,149.258
C01610=1116.670,4.902,-51.449,179.747,6.491,149.259
C01611=1116.665,5.151,-51.463,179.747,6.495,149.260
C01612=1116.660,5.400,-51.477,179.748,6.500,149.260
C01613=1116.655,5.650,-51.492,179.748,6.504,149.261
C01614=1116.650,5.900,-51.506,179.749,6.508,149.262
C01615=1116.645,6.150,-51.520,179.749,6.513,149.263
C01616=1116.639,6.399,-51.534,179.750,6.518,149.264
C01617=1116.634,6.648,-51.548,179.751,6.522,149.264
C01618=1116.629,6.898,-51.563,179.751,6.527,149.265
C01619=1116.624,7.148,-51.577,179.752,6.532,149.266
C01620=1116.619,7.397,-51.591,179.752,6.536,149.267
C01621=1116.614,7.646,-51.605,179.752,6.540,149.268
C01622=1116.609,7.896,-51.619,179.753,6.545,149.269
C01623=1116.604,8.146,-51.634,179.753,6.550,149.270
C01624=1116.599,8.396,-51.648,179.754,6.554,149.271
C01625=1116.594,8.610,-51.660,179.755,6.559,149.271
C01626=1116.590,8.825,-51.672,179.755,6.562,149.272
C01627=1116.586,9.040,-51.685,179.756,6.566,149.273
C01628=1116.581,9.254,-51.697,179.756,6.571,149.273
C01629=1116.577,9.468,-51.709,179.757,6.574,149.274
C01630=1116.572,9.684,-51.721,179.758,6.578,149.275
C01631=1116.568,9.898,-51.733,179.758,6.582,149.275
C01632=1116.564,10.112,-51.746,179.758,6.586,149.276
C01633=1116.559,10.362,-51.760,179.759,6.590,149.277
C01634=1116.554,10.612,-51.774,179.760,6.595,149.278
C01635=1116.549,10.861,-51.788,179.760,6.600,149.279
C01636=1116.544,11.110,-51.803,179.761,6.604,149.280
C01637=1116.538,11.360,-51.818,179.762,6.609,149.280
C01638=1116.533,11.610,-51.832,179.762,6.613,149.281
C01639=1116.528,11.859,-51.847,179.763,6.618,149.282
C01640=1116.523,12.109,-51.861,179.764,6.622,149.283
C01641=1116.518,12.359,-51.875,179.765,6.627,149.284
C01642=1116.513,12.607,-51.890,179.765,6.632,149.284
C01643=1116.508,12.857,-51.904,179.766,6.636,149.285
C01644=1116.503,13.107,-51.918,179.767,6.641,149.286
C01645=1116.498,13.356,-51.933,179.767,6.646,149.287
C01646=1116.493,13.606,-51.948,179.768,6.650,149.288
C01647=1116.488,13.855,-51.963,179.769,6.655,149.288
C01648=1116.483,14.105,-51.977,179.769,6.659,149.289
C01649=1116.478,14.355,-51.991,179.770,6.664,149.290
C01650=1116.473,14.604,-52.006,179.771,6.668,149.291
C01651=1116.468,14.853,-52.020,179.772,6.673,149.292
C01652=1116.462,15.103,-52.035,179.773,6.677,149.292
C01653=1116.457,15.353,-52.049,179.772,6.681,149.293
C01654=1116.453,15.602,-52.064,179.774,6.686,149.294
C01655=1116.448,15.852,-52.078,179.774,6.690,149.295
C01656=1116.443,16.101,-52.093,179.775,6.695,149.295
C01657=1116.437,16.351,-52.108,179.776,6.699,149.296
C01658=1116.432,16.600,-52.123,179.777,6.704,149.297
C01659=1116.428,16.849,-52.138,179.777,6.708,149.298
C01660=1116.423,17.099,-52.152,179.778,6.713,149.299
C01661=1116.417,17.349,-52.167,179.779,6.717,149.299
C01662=1116.412,17.598,-52.182,179.780,6.722,149.300
C01663=1116.407,17.848,-52.196,179.780,6.726,149.301
C01664=1116.403,18.097,-52.211,179.782,6.731,149.302
C01665=1116.397,18.347,-52.226,179.782,6.735,149.302
C01666=1116.392,18.597,-52.240,179.783,6.740,149.303
C01667=1116.387,18.846,-52.255,179.783,6.744,149.304
C01668=1116.382,19.096,-52.269,179.784,6.748,149.305
C01669=1116.377,19.345,-52.285,179.785,6.753,149.306
C01670=1116.372,19.595,-52.299,179.786,6.757,149.306
C01671=1116.368,19.844,-52.314,179.787,6.761,149.307
C01672=1116.362,20.094,-52.329,179.787,6.766,149.308
C01673=1116.357,20.343,-52.344,179.788,6.770,149.308
C01674=1116.352,20.593,-52.358,179.789,6.775,149.309
C01675=1116.347,20.842,-52.374,179.790,6.779,149.310
C01676=1116.342,21.092,-52.388,179.791,6.784,149.311
C01677=1116.337,21.341,-52.403,179.792,6.788,149.311
C01678=1116.332,21.591,-52.418,179.793,6.793,149.312
C01679=1116.327,21.840,-52.433,179.793,6.797,149.313
C01680=1116.321,22.089,-52.449,179.794,6.801,149.314
C01681=1116.318,22.304,-52.461,179.795,6.805,149.314
C01682=1116.313,22.519,-52.474,179.795,6.809,149.315
C01683=1116.309,22.733,-52.486,179.796,6.812,149.315
C01684=1116.304,22.948,-52.499,179.797,6.816,149.316
C01685=1116.300,23.162,-52.512,179.797,6.820,149.317
C01686=1116.296,23.377,-52.525,179.799,6.824,149.317
C01687=1116.291,23.592,-52.538,179.799,6.828,149.318
C01688=1116.288,23.806,-52.551,179.799,6.831,149.319
C01689=1116.282,24.056,-52.566,179.800,6.835,149.319
C01690=1116.277,24.305,-52.581,179.801,6.840,149.320
C01691=1116.272,24.554,-52.597,179.802,6.844,149.321
C01692=1116.267,24.804,-52.611,179.803,6.849,149.322
C01693=1116.262,25.053,-52.627,179.804,6.853,149.322
C01694=1116.257,25.302,-52.642,179.805,6.857,149.323
C01695=1116.251,25.552,-52.657,179.805,6.861,149.324
C01696=1116.247,25.802,-52.672,179.806,6.866,149.324
C01697=1116.242,26.051,-52.686,179.807,6.870,149.325
C01698=1116.237,26.301,-52.702,179.808,6.874,149.326
C01699=1116.232,26.550,-52.717,179.809,6.879,149.326
C01700=1116.227,26.800,-52.732,179.810,6.883,149.327
C01701=1116.222,27.049,-52.747,179.811,6.888,149.328
C01702=1116.217,27.298,-52.763,179.812,6.892,149.328
C01703=1116.211,27.548,-52.778,179.813,6.896,149.329
C01704=1116.206,27.797,-52.793,179.814,6.900,149.330
C01705=1116.202,28.048,-52.809,179.814,6.904,149.331
C01706=1116.197,28.297,-52.824,179.815,6.909,149.331
C01707=1116.192,28.546,-52.839,179.816,6.913,149.332
C01708=1116.187,28.796,-52.854,179.817,6.917,149.333
C01709=1116.181,29.045,-52.869,179.818,6.922,149.333
C01710=1116.177,29.294,-52.884,179.819,6.926,149.334
C01711=1116.172,29.544,-52.900,179.820,6.930,149.335
C01712=1116.166,29.794,-52.916,179.822,6.935,149.335
C01713=1116.162,30.043,-52.931,179.822,6.939,149.336
C01714=1116.156,30.292,-52.946,179.823,6.943,149.337
C01715=1116.152,30.541,-52.961,179.824,6.947,149.337
C01716=1116.147,30.791,-52.977,179.825,6.951,149.338
C01717=1116.141,31.042,-52.992,179.826,6.956,149.339
C01718=1116.137,31.291,-53.007,179.827,6.960,149.339
C01719=1116.131,31.540,-53.023,179.828,6.964,149.340
C01720=1116.126,31.789,-53.038,179.829,6.969,149.341
C01721=1116.122,32.039,-53.054,179.829,6.972,149.341
C01722=1116.116,32.289,-53.069,179.830,6.977,149.342
C01723=1116.111,32.538,-53.085,179.831,6.981,149.343
C01724=1116.106,32.787,-53.100,179.833,6.985,149.343
C01725=1116.102,33.037,-53.116,179.834,6.989,149.344
C01726=1116.096,33.287,-53.131,179.835,6.994,149.345
C01727=1116.092,33.536,-53.146,179.836,6.998,149.345
C01728=1116.086,33.785,-53.162,179.837,7.002,149.346
C01729=1116.081,34.035,-53.178,179.837,7.006,149.347
C01730=1116.077,34.284,-53.193,179.838,7.010,149.347
C01731=1116.072,34.533,-53.209,179.839,7.015,149.348
C01732=1116.066,34.782,-53.225,179.840,7.019,149.349
C01733=1116.061,35.033,-53.241,179.842,7.023,149.349
C01734=1116.057,35.282,-53.256,179.843,7.027,149.350
C01735=1116.051,35.531,-53.271,179.844,7.032,149.350
C01736=1116.047,35.781,-53.287,179.844,7.035,149.351
C01737=1116.040,36.105,-53.307,179.846,7.042,149.352
C01738=1116.033,36.430,-53.328,179.847,7.047,149.353
C01739=1116.027,36.754,-53.348,179.849,7.052,149.354
C01740=1116.020,37.078,-53.368,179.850,7.058,149.354
C01741=1116.013,37.432,-53.391,179.851,7.063,149.355
C01742=1116.006,37.786,-53.414,179.853,7.070,149.356
C01743=1115.999,38.140,-53.435,179.854,7.075,149.357
C01744=1115.992,38.494,-53.458,179.856,7.082,149.358
C01745=1115.987,38.743,-53.473,179.856,7.085,149.359
C01746=1115.982,38.994,-53.489,179.858,7.089,149.359
C01747=1115.977,39.242,-53.506,179.859,7.093,149.360
C01748=1115.972,39.492,-53.521,179.860,7.098,149.360
C01749=1115.967,39.742,-53.537,179.861,7.102,149.361
C01750=1115.962,39.991,-53.553,179.862,7.106,149.362
C01751=1115.957,40.241,-53.569,179.863,7.110,149.362
C01752=1115.953,40.490,-53.584,179.863,7.114,149.363
C01753=1115.947,40.739,-53.600,179.865,7.118,149.364
C01754=1115.943,40.989,-53.617,179.866,7.122,149.364
C01755=1115.937,41.238,-53.632,179.867,7.127,149.365
C01756=1115.933,41.488,-53.648,179.868,7.131,149.365
C01757=1115.927,41.737,-53.664,179.869,7.135,149.366
C01758=1115.922,41.986,-53.680,179.871,7.139,149.367
C01759=1115.918,42.236,-53.697,179.871,7.143,149.367
C01760=1115.912,42.485,-53.712,179.872,7.147,149.368
C01761=1115.907,42.735,-53.728,179.873,7.151,149.369
C01762=1115.902,42.984,-53.745,179.875,7.155,149.369
C01763=1115.898,43.234,-53.761,179.876,7.159,149.370
C01764=1115.892,43.483,-53.777,179.877,7.164,149.370
C01765=1115.887,43.732,-53.792,179.878,7.168,149.371
C01766=1115.883,43.982,-53.809,179.879,7.171,149.371
C01767=1115.877,44.231,-53.825,179.880,7.175,149.372
C01768=1115.873,44.481,-53.841,179.881,7.180,149.373
C01769=1115.867,44.730,-53.857,179.882,7.184,149.373
C01770=1115.863,44.980,-53.873,179.884,7.188,149.374
C01771=1115.857,45.229,-53.889,179.885,7.192,149.374
C01772=1115.853,45.479,-53.906,179.886,7.197,149.375
C01773=1115.848,45.728,-53.921,179.887,7.200,149.376
C01774=1115.843,45.978,-53.938,179.888,7.204,149.376
C01775=1115.838,46.227,-53.954,179.889,7.208,149.377
C01776=1115.833,46.476,-53.970,179.890,7.213,149.377
C01777=1115.828,46.726,-53.986,179.892,7.217,149.378
C01778=1115.823,46.975,-54.003,179.893,7.221,149.378
C01779=1115.818,47.225,-54.018,179.894,7.225,149.379
C01780=1115.814,47.474,-54.035,179.895,7.228,149.380
C01781=1115.808,47.723,-54.051,179.896,7.233,149.380
C01782=1115.804,47.973,-54.067,179.897,7.237,149.381
C01783=1115.799,48.222,-54.083,179.899,7.241,149.381
C01784=1115.793,48.472,-54.101,179.900,7.245,149.382
C01785=1115.788,48.721,-54.116,179.901,7.249,149.383
C01786=1115.784,48.971,-54.133,179.902,7.253,149.383
C01787=1115.779,49.220,-54.150,179.903,7.257,149.384
C01788=1115.774,49.469,-54.165,179.904,7.261,149.384
C01789=1115.769,49.684,-54.179,179.905,7.265,149.385
C01790=1115.765,49.897,-54.193,179.906,7.268,149.385
C01791=1115.761,50.113,-54.208,179.907,7.271,149.386
C01792=1115.757,50.327,-54.222,179.908,7.276,149.386
C01793=1115.752,50.541,-54.235,179.909,7.279,149.387
C01794=1115.748,50.755,-54.250,179.910,7.282,149.387
C01795=1115.744,50.971,-54.265,179.912,7.286,149.388
C01796=1115.740,51.185,-54.278,179.912,7.289,149.388
C01797=1115.735,51.434,-54.295,179.914,7.293,149.389
C01798=1115.730,51.683,-54.311,179.915,7.297,149.389
C01799=1115.726,51.933,-54.328,179.916,7.301,149.390
C01800=1115.719,52.182,-54.344,179.917,7.305,149.390
C01801=1115.715,52.432,-54.361,179.919,7.309,149.391
C01802=1115.710,52.681,-54.377,179.920,7.313,149.391
C01803=1115.705,52.930,-54.394,179.921,7.317,149.392
C01804=1115.700,53.180,-54.411,179.922,7.321,149.393
C01805=1115.695,53.429,-54.427,179.923,7.326,149.393
C01806=1115.690,53.679,-54.443,179.924,7.329,149.394
C01807=1115.685,53.928,-54.460,179.925,7.333,149.394
C01808=1115.680,54.177,-54.477,179.927,7.337,149.395
C01809=1115.676,54.427,-54.493,179.928,7.341,149.395
C01810=1115.670,54.676,-54.510,179.930,7.345,149.396
C01811=1115.665,54.925,-54.527,179.931,7.349,149.396
C01812=1115.661,55.175,-54.544,179.932,7.353,149.397
C01813=1115.656,55.424,-54.560,179.933,7.358,149.398
C01814=1115.650,55.673,-54.577,179.934,7.361,149.398
C01815=1115.646,55.923,-54.594,179.935,7.365,149.399
C01816=1115.641,56.172,-54.610,179.936,7.369,149.399
C01817=1115.636,56.421,-54.627,179.938,7.373,149.400
C01818=1115.631,56.672,-54.643,179.939,7.378,149.400
C01819=1115.626,56.920,-54.660,179.941,7.381,149.401
C01820=1115.621,57.170,-54.677,179.942,7.385,149.401
C01821=1115.616,57.419,-54.694,179.943,7.389,149.402
C01822=1115.612,57.669,-54.711,179.944,7.393,149.402
C01823=1115.606,57.918,-54.728,179.945,7.397,149.403
C01824=1115.602,58.167,-54.745,179.947,7.401,149.403
C01825=1115.596,58.417,-54.762,179.948,7.405,149.404
C01826=1115.592,58.666,-54.779,179.950,7.409,149.404
C01827=1115.586,58.915,-54.795,179.951,7.414,149.405
C01828=1115.582,59.165,-54.812,179.952,7.417,149.406
C01829=1115.577,59.414,-54.829,179.953,7.421,149.406
C01830=1115.571,59.664,-54.846,179.954,7.425,149.407
C01831=1115.567,59.913,-54.862,179.955,7.429,149.407
C01832=1115.562,60.163,-54.880,179.957,7.433,149.408
C01833=1115.557,60.412,-54.896,179.958,7.437,149.408
C01834=1115.552,60.661,-54.914,179.960,7.441,149.409
C01835=1115.547,60.910,-54.931,179.961,7.445,149.409
C01836=1115.542,61.160,-54.948,179.962,7.449,149.410
C01837=1115.537,61.410,-54.965,179.963,7.453,149.410
C01838=1115.532,61.659,-54.982,179.964,7.457,149.411
C01839=1115.528,61.907,-54.999,179.966,7.461,149.411
C01840=1115.522,62.157,-55.016,179.967,7.465,149.412
C01841=1115.518,62.407,-55.033,179.969,7.469,149.412
C01842=1115.513,62.657,-55.050,179.970,7.473,149.413
C01843=1115.508,62.906,-55.067,179.971,7.477,149.413
C01844=1115.503,63.155,-55.085,179.973,7.481,149.414
C01845=1115.499,63.370,-55.098,179.974,7.484,149.414
C01846=1115.494,63.584,-55.113,179.975,7.487,149.415
C01847=1115.491,63.798,-55.128,179.976,7.491,149.415
C01848=1115.486,64.012,-55.143,179.977,7.494,149.416
C01849=1115.482,64.226,-55.158,179.978,7.497,149.416
